C01813=1053.237,59.929,422.366,171.034,32.293,156.055
C01814=1053.230,59.680,422.384,171.032,32.290,156.054
C01815=1053.224,59.431,422.401,171.030,32.288,156.054
C01816=1053.217,59.181,422.419,171.029,32.286,156.054
C01817=1053.211,58.932,422.435,171.027,32.284,156.053
C01818=1053.205,58.682,422.453,171.025,32.282,156.053
C01819=1053.199,58.433,422.470,171.024,32.280,156.053
C01820=1053.193,58.184,422.488,171.022,32.278,156.052
C01821=1053.187,57.935,422.505,171.020,32.276,156.052
C01822=1053.180,57.685,422.522,171.019,32.273,156.052
C01823=1053.174,57.436,422.539,171.017,32.271,156.051
C01824=1053.168,57.186,422.556,171.015,32.269,156.051
C01825=1053.162,56.937,422.574,171.014,32.267,156.051
C01826=1053.155,56.688,422.591,171.012,32.264,156.050
C01827=1053.149,56.439,422.608,171.010,32.262,156.050
C01828=1053.143,56.189,422.625,171.010,32.260,156.050
C01829=1053.137,55.940,422.642,171.008,32.258,156.049
C01830=1053.131,55.690,422.660,171.006,32.256,156.049
C01831=1053.125,55.442,422.677,171.005,32.254,156.049
C01832=1053.118,55.191,422.694,171.003,32.252,156.048
C01833=1053.113,54.942,422.711,171.001,32.250,156.048
C01834=1053.106,54.694,422.728,171.000,32.247,156.048
C01835=1053.099,54.444,422.746,170.998,32.245,156.047
C01836=1053.094,54.195,422.762,170.996,32.243,156.047
C01837=1053.087,53.945,422.780,170.995,32.241,156.047
C01838=1053.082,53.696,422.797,170.993,32.238,156.046
C01839=1053.075,53.446,422.814,170.991,32.236,156.046
C01840=1053.069,53.197,422.831,170.990,32.234,156.046
C01841=1053.063,52.948,422.849,170.988,32.232,156.045
C01842=1053.057,52.699,422.866,170.987,32.230,156.045
C01843=1053.051,52.450,422.882,170.986,32.228,156.045
C01844=1053.045,52.200,422.900,170.984,32.226,156.044
C01845=1053.039,51.950,422.916,170.983,32.223,156.044
C01846=1053.032,51.701,422.934,170.981,32.221,156.044
C01847=1053.026,51.452,422.951,170.979,32.219,156.043
C01848=1053.020,51.203,422.967,170.978,32.216,156.043
C01849=1053.013,50.953,422.985,170.976,32.214,156.043
C01850=1053.008,50.704,423.002,170.974,32.212,156.042
C01851=1053.002,50.455,423.019,170.973,32.210,156.042
C01852=1052.995,50.205,423.036,170.971,32.208,156.041
C01853=1052.990,49.956,423.053,170.969,32.206,156.041
C01854=1052.983,49.706,423.070,170.968,32.204,156.041
C01855=1052.977,49.457,423.086,170.966,32.201,156.040
C01856=1052.972,49.208,423.104,170.964,32.199,156.040
C01857=1052.965,48.958,423.121,170.964,32.197,156.040
C01858=1052.959,48.709,423.138,170.962,32.195,156.040
C01859=1052.953,48.460,423.155,170.960,32.192,156.039
C01860=1052.947,48.210,423.172,170.959,32.190,156.039
C01861=1052.940,47.961,423.189,170.957,32.188,156.039
C01862=1052.935,47.712,423.206,170.955,32.186,156.038
C01863=1052.928,47.462,423.223,170.954,32.184,156.038
C01864=1052.922,47.213,423.239,170.952,32.182,156.037
C01865=1052.917,46.964,423.257,170.950,32.179,156.037
C01866=1052.911,46.714,423.273,170.949,32.177,156.037
C01867=1052.904,46.465,423.290,170.947,32.175,156.036
C01868=1052.899,46.215,423.307,170.945,32.173,156.036
C01869=1052.891,45.930,423.327,170.944,32.170,156.036
C01870=1052.885,45.644,423.345,170.942,32.168,156.035
C01871=1052.877,45.358,423.365,170.941,32.165,156.035
C01872=1052.870,45.072,423.385,170.939,32.162,156.034
C01873=1052.864,44.823,423.401,170.937,32.160,156.034
C01874=1052.859,44.573,423.418,170.936,32.158,156.034
C01875=1052.853,44.325,423.435,170.934,32.156,156.033
C01876=1052.846,44.075,423.451,170.932,32.154,156.033
C01877=1052.841,43.826,423.469,170.931,32.152,156.033
C01878=1052.835,43.576,423.485,170.929,32.149,156.032
C01879=1052.828,43.326,423.502,170.927,32.147,156.032
C01880=1052.822,43.077,423.519,170.926,32.145,156.032
C01881=1052.816,42.828,423.535,170.924,32.143,156.032
C01882=1052.810,42.579,423.551,170.922,32.141,156.031
C01883=1052.803,42.329,423.569,170.921,32.138,156.031
C01884=1052.797,42.080,423.585,170.920,32.136,156.030
C01885=1052.791,41.831,423.601,170.918,32.134,156.030
C01886=1052.785,41.581,423.619,170.917,32.132,156.030
C01887=1052.779,41.332,423.635,170.915,32.130,156.030
C01888=1052.773,41.082,423.651,170.913,32.128,156.029
C01889=1052.767,40.833,423.669,170.911,32.125,156.029
C01890=1052.761,40.583,423.685,170.910,32.123,156.029
C01891=1052.755,40.334,423.701,170.908,32.121,156.028
C01892=1052.749,40.085,423.718,170.906,32.119,156.028
C01893=1052.743,39.836,423.735,170.905,32.117,156.028
C01894=1052.736,39.586,423.751,170.903,32.115,156.027
C01895=1052.730,39.337,423.768,170.901,32.113,156.027
C01896=1052.724,39.087,423.784,170.900,32.111,156.027
C01897=1052.718,38.838,423.800,170.899,32.109,156.026
C01898=1052.712,38.589,423.817,170.897,32.106,156.026
C01899=1052.705,38.339,423.834,170.896,32.104,156.026
C01900=1052.699,38.090,423.850,170.894,32.102,156.025
C01901=1052.693,37.840,423.866,170.892,32.100,156.025
C01902=1052.687,37.591,423.882,170.891,32.098,156.025
C01903=1052.681,37.342,423.900,170.889,32.096,156.024
C01904=1052.675,37.092,423.916,170.887,32.093,156.024
C01905=1052.669,36.843,423.932,170.886,32.091,156.024
C01906=1052.662,36.594,423.948,170.884,32.089,156.023
C01907=1052.656,36.345,423.964,170.882,32.087,156.023
C01908=1052.649,36.094,423.981,170.881,32.085,156.023
C01909=1052.644,35.845,423.997,170.879,32.083,156.022
C01910=1052.638,35.596,424.013,170.878,32.081,156.022
C01911=1052.632,35.346,424.030,170.876,32.079,156.022
C01912=1052.624,35.097,424.046,170.875,32.077,156.022
C01913=1052.618,34.848,424.063,170.873,32.075,156.021
C01914=1052.612,34.599,424.079,170.871,32.072,156.021
C01915=1052.606,34.349,424.095,170.870,32.070,156.021
C01916=1052.600,34.100,424.111,170.868,32.068,156.020
C01917=1052.594,33.851,424.127,170.866,32.066,156.020
C01918=1052.587,33.601,424.144,170.865,32.064,156.020
C01919=1052.581,33.351,424.160,170.863,32.062,156.019
C01920=1052.575,33.102,424.176,170.861,32.060,156.019
C01921=1052.569,32.853,424.192,170.860,32.058,156.019
C01922=1052.563,32.603,424.209,170.858,32.056,156.018
C01923=1052.556,32.354,424.224,170.857,32.053,156.018
C01924=1052.550,32.104,424.241,170.855,32.051,156.018
C01925=1052.544,31.855,424.257,170.854,32.049,156.017
C01926=1052.538,31.606,424.273,170.852,32.047,156.017
C01927=1052.532,31.356,424.290,170.850,32.045,156.017
C01928=1052.525,31.107,424.305,170.849,32.043,156.017
C01929=1052.519,30.858,424.322,170.847,32.041,156.016
C01930=1052.513,30.609,424.338,170.845,32.039,156.016
C01931=1052.508,30.359,424.354,170.844,32.037,156.015
C01932=1052.501,30.109,424.371,170.842,32.035,156.015
C01933=1052.494,29.824,424.389,170.840,32.032,156.015
C01934=1052.487,29.538,424.407,170.838,32.030,156.014
C01935=1052.480,29.252,424.426,170.837,32.028,156.014
C01936=1052.474,28.966,424.444,170.835,32.025,156.014
C01937=1052.467,28.717,424.459,170.833,32.023,156.014
C01938=1052.461,28.467,424.475,170.832,32.021,156.013
C01939=1052.454,28.217,424.492,170.830,32.019,156.013
C01940=1052.448,27.968,424.508,170.828,32.017,156.013
C01941=1052.442,27.719,424.524,170.827,32.015,156.012
C01942=1052.436,27.470,424.540,170.825,32.013,156.012
C01943=1052.429,27.220,424.555,170.823,32.011,156.012
C01944=1052.423,26.971,424.571,170.821,32.009,156.011
C01945=1052.417,26.721,424.588,170.820,32.006,156.011
C01946=1052.411,26.472,424.603,170.818,32.004,156.011
C01947=1052.405,26.223,424.620,170.817,32.002,156.010
C01948=1052.398,25.973,424.635,170.816,32.000,156.010
C01949=1052.392,25.723,424.651,170.814,31.998,156.010
C01950=1052.385,25.474,424.667,170.812,31.996,156.009
C01951=1052.379,25.225,424.683,170.810,31.994,156.009
C01952=1052.374,24.975,424.699,170.809,31.992,156.009
C01953=1052.367,24.726,424.714,170.807,31.990,156.009
C01954=1052.361,24.476,424.731,170.805,31.988,156.008
C01955=1052.354,24.227,424.746,170.804,31.986,156.008
C01956=1052.349,23.977,424.762,170.802,31.984,156.008
C01957=1052.342,23.728,424.777,170.800,31.982,156.007
C01958=1052.336,23.479,424.794,170.798,31.979,156.007
C01959=1052.330,23.229,424.809,170.798,31.978,156.007
C01960=1052.324,22.980,424.825,170.796,31.975,156.006
C01961=1052.318,22.731,424.841,170.794,31.973,156.006
C01962=1052.311,22.481,424.856,170.793,31.971,156.006
C01963=1052.305,22.232,424.872,170.791,31.969,156.006
C01964=1052.299,21.983,424.888,170.789,31.967,156.005
C01965=1052.293,21.733,424.904,170.787,31.965,156.005
C01966=1052.286,21.484,424.919,170.786,31.963,156.005
C01967=1052.280,21.234,424.936,170.784,31.961,156.004
C01968=1052.275,20.984,424.951,170.782,31.959,156.004
C01969=1052.268,20.735,424.967,170.781,31.957,156.004
C01970=1052.262,20.485,424.982,170.779,31.955,156.003
C01971=1052.256,20.236,424.998,170.778,31.953,156.003
C01972=1052.250,19.987,425.014,170.776,31.951,156.003
C01973=1052.243,19.737,425.029,170.775,31.949,156.003
C01974=1052.237,19.488,425.045,170.773,31.947,156.002
C01975=1052.231,19.238,425.060,170.771,31.945,156.002
C01976=1052.224,18.989,425.076,170.769,31.943,156.002
C01977=1052.219,18.739,425.092,170.768,31.941,156.001
C01978=1052.212,18.490,425.107,170.766,31.939,156.001
C01979=1052.206,18.240,425.123,170.764,31.937,156.001
C01980=1052.200,17.991,425.138,170.762,31.934,156.001
C01981=1052.193,17.741,425.153,170.761,31.933,156.000
C01982=1052.187,17.492,425.170,170.760,31.930,156.000
C01983=1052.181,17.242,425.185,170.758,31.928,156.000
C01984=1052.175,16.993,425.201,170.757,31.926,155.999
C01985=1052.169,16.743,425.216,170.755,31.924,155.999
C01986=1052.162,16.494,425.231,170.753,31.922,155.999
C01987=1052.156,16.244,425.247,170.751,31.920,155.998
C01988=1052.150,15.996,425.262,170.750,31.918,155.998
C01989=1052.144,15.746,425.277,170.748,31.916,155.998
C01990=1052.138,15.497,425.293,170.746,31.914,155.998
C01991=1052.131,15.247,425.308,170.744,31.913,155.997
C01992=1052.126,14.998,425.325,170.743,31.911,155.997
C01993=1052.119,14.748,425.340,170.741,31.909,155.997
C01994=1052.113,14.499,425.355,170.740,31.906,155.996
C01995=1052.107,14.249,425.371,170.738,31.904,155.996
C01996=1052.100,14.000,425.386,170.737,31.902,155.996
C01997=1052.094,13.715,425.403,170.735,31.900,155.996
C01998=1052.087,13.431,425.420,170.733,31.898,155.995
C01999=1052.079,13.146,425.439,170.731,31.896,155.995
C02000=1052.071,12.862,425.455,170.729,31.893,155.995
C02001=1052.065,12.612,425.471,170.727,31.891,155.994
C02002=1052.059,12.362,425.486,170.725,31.889,155.994
C02003=1052.052,12.113,425.502,170.723,31.887,155.994
C02004=1052.046,11.864,425.517,170.722,31.886,155.994
C02005=1052.040,11.615,425.531,170.721,31.884,155.993
C02006=1052.034,11.365,425.546,170.719,31.882,155.993
C02007=1052.027,11.116,425.562,170.717,31.880,155.993
C02008=1052.021,10.866,425.577,170.715,31.877,155.992
C02009=1052.015,10.616,425.592,170.714,31.876,155.992
C02010=1052.009,10.367,425.607,170.712,31.874,155.992
C02011=1052.002,10.118,425.623,170.710,31.872,155.992
C02012=1051.996,9.868,425.638,170.708,31.870,155.991
C02013=1051.989,9.618,425.653,170.707,31.868,155.991
C02014=1051.983,9.369,425.667,170.705,31.866,155.991
C02015=1051.977,9.120,425.684,170.703,31.864,155.990
C02016=1051.971,8.870,425.699,170.702,31.862,155.990
C02017=1051.965,8.621,425.713,170.701,31.860,155.990
C02018=1051.958,8.371,425.728,170.699,31.858,155.990
C02019=1051.952,8.121,425.743,170.697,31.856,155.989
C02020=1051.945,7.872,425.759,170.695,31.854,155.989
C02021=1051.939,7.623,425.774,170.693,31.852,155.989
C02022=1051.933,7.374,425.789,170.692,31.851,155.989
C02023=1051.927,7.124,425.803,170.690,31.848,155.988
C02024=1051.921,6.874,425.819,170.688,31.846,155.988
C02025=1051.915,6.625,425.834,170.686,31.844,155.988
C02026=1051.909,6.376,425.849,170.685,31.842,155.987
C02027=1051.902,6.127,425.864,170.684,31.840,155.987
C02028=1051.896,5.877,425.879,170.682,31.839,155.987
C02029=1051.889,5.627,425.894,170.680,31.837,155.987
C02030=1051.883,5.378,425.909,170.678,31.835,155.986
C02031=1051.877,5.129,425.924,170.677,31.833,155.986
C02032=1051.871,4.879,425.939,170.675,31.831,155.986
C02033=1051.865,4.629,425.954,170.673,31.828,155.985
C02034=1051.859,4.379,425.969,170.671,31.827,155.985
C02035=1051.853,4.130,425.984,170.670,31.825,155.985
C02036=1051.847,3.881,425.999,170.668,31.823,155.985
C02037=1051.840,3.631,426.014,170.666,31.821,155.984
C02038=1051.834,3.381,426.028,170.665,31.819,155.984
C02039=1051.828,3.132,426.043,170.663,31.817,155.984
C02040=1051.821,2.883,426.059,170.662,31.815,155.984
C02041=1051.815,2.634,426.074,170.660,31.813,155.983
C02042=1051.809,2.384,426.089,170.658,31.811,155.983
C02043=1051.803,2.135,426.103,170.656,31.809,155.983
C02044=1051.797,1.885,426.118,170.654,31.807,155.982
C02045=1051.790,1.636,426.133,170.653,31.806,155.982
C02046=1051.784,1.386,426.147,170.651,31.803,155.982
C02047=1051.778,1.137,426.162,170.649,31.801,155.982
C02048=1051.772,0.887,426.177,170.648,31.799,155.981
C02049=1051.766,0.637,426.192,170.647,31.797,155.981
C02050=1051.760,0.388,426.207,170.645,31.795,155.981
C02051=1051.754,0.138,426.222,170.643,31.794,155.981
C02052=1051.748,-0.111,426.237,170.641,31.792,155.980
C02053=1051.742,-0.360,426.251,170.639,31.790,155.980
C02054=1051.736,-0.610,426.266,170.638,31.788,155.980
C02055=1051.729,-0.860,426.281,170.636,31.785,155.979
C02056=1051.723,-1.109,426.296,170.634,31.784,155.979
C02057=1051.717,-1.358,426.311,170.632,31.782,155.979
C02058=1051.711,-1.608,426.326,170.630,31.780,155.979
C02059=1051.705,-1.857,426.340,170.630,31.778,155.978
C02060=1051.699,-2.107,426.355,170.628,31.776,155.978
C02061=1051.692,-2.389,426.371,170.626,31.774,155.978
C02062=1051.685,-2.672,426.388,170.624,31.772,155.977
C02063=1051.678,-2.954,426.405,170.622,31.769,155.977
C02064=1051.671,-3.238,426.421,170.620,31.767,155.977
C02065=1051.665,-3.487,426.436,170.618,31.765,155.977
C02066=1051.659,-3.736,426.451,170.616,31.763,155.976
C02067=1051.652,-3.986,426.466,170.614,31.761,155.976
C02068=1051.646,-4.235,426.479,170.612,31.760,155.976
C02069=1051.640,-4.485,426.494,170.611,31.757,155.976
C02070=1051.633,-4.735,426.509,170.610,31.756,155.975
C02071=1051.627,-4.983,426.524,170.608,31.754,155.975
C02072=1051.621,-5.233,426.537,170.606,31.752,155.975
C02073=1051.614,-5.483,426.552,170.604,31.750,155.975
C02074=1051.608,-5.732,426.567,170.602,31.748,155.974
C02075=1051.602,-5.982,426.580,170.601,31.746,155.974
C02076=1051.595,-6.232,426.595,170.599,31.745,155.974
C02077=1051.589,-6.481,426.610,170.597,31.743,155.974
C02078=1051.583,-6.730,426.625,170.595,31.741,155.973
C02079=1051.577,-6.980,426.638,170.594,31.739,155.973
C02080=1051.570,-7.229,426.653,170.592,31.737,155.973
C02081=1051.564,-7.479,426.668,170.591,31.736,155.973
C02082=1051.559,-7.728,426.682,170.589,31.734,155.972
C02083=1051.552,-7.978,426.696,170.587,31.732,155.972
C02084=1051.545,-8.227,426.711,170.585,31.730,155.972
C02085=1051.540,-8.477,426.725,170.583,31.728,155.972
C02086=1051.533,-8.726,426.739,170.581,31.726,155.971
C02087=1051.527,-8.976,426.753,170.579,31.724,155.971
C02088=1051.521,-9.226,426.768,170.578,31.722,155.971
C02089=1051.515,-9.475,426.783,170.576,31.721,155.971
C02090=1051.508,-9.725,426.796,170.575,31.719,155.970
C02091=1051.502,-9.974,426.811,170.573,31.717,155.970
C02092=1051.496,-10.224,426.825,170.571,31.715,155.970
C02093=1051.489,-10.473,426.840,170.569,31.713,155.970
C02094=1051.483,-10.722,426.854,170.568,31.712,155.969
C02095=1051.477,-10.972,426.868,170.566,31.710,155.969
C02096=1051.471,-11.221,426.882,170.564,31.708,155.969
C02097=1051.465,-11.471,426.897,170.562,31.706,155.969
C02098=1051.459,-11.720,426.911,170.560,31.704,155.968
C02099=1051.452,-11.970,426.925,170.558,31.702,155.968
C02100=1051.446,-12.220,426.940,170.557,31.700,155.968
C02101=1051.440,-12.469,426.954,170.556,31.698,155.968
C02102=1051.433,-12.719,426.968,170.554,31.697,155.967
C02103=1051.428,-12.968,426.982,170.552,31.695,155.967
C02104=1051.421,-13.218,426.997,170.550,31.693,155.967
C02105=1051.415,-13.467,427.010,170.548,31.691,155.967
C02106=1051.409,-13.717,427.025,170.546,31.689,155.966
C02107=1051.403,-13.966,427.039,170.545,31.688,155.966
C02108=1051.396,-14.216,427.053,170.543,31.686,155.966
C02109=1051.391,-14.465,427.067,170.541,31.684,155.966
C02110=1051.384,-14.716,427.081,170.540,31.682,155.965
C02111=1051.378,-14.964,427.095,170.538,31.680,155.965
C02112=1051.372,-15.215,427.110,170.536,31.678,155.965
C02113=1051.365,-15.463,427.124,170.534,31.676,155.965
C02114=1051.359,-15.714,427.138,170.532,31.675,155.965
C02115=1051.353,-15.963,427.151,170.531,31.673,155.964
C02116=1051.347,-16.212,427.166,170.529,31.671,155.964
C02117=1051.340,-16.462,427.179,170.527,31.669,155.964
C02118=1051.334,-16.712,427.194,170.525,31.668,155.964
C02119=1051.328,-16.961,427.208,170.523,31.666,155.963
C02120=1051.322,-17.211,427.222,170.522,31.664,155.963
C02121=1051.316,-17.460,427.235,170.520,31.663,155.963
C02122=1051.308,-17.710,427.249,170.518,31.661,155.963
C02123=1051.303,-17.959,427.263,170.517,31.659,155.962
C02124=1051.297,-18.208,427.277,170.515,31.657,155.962
C02125=1051.290,-18.489,427.292,170.513,31.656,155.962
C02126=1051.283,-18.771,427.308,170.510,31.653,155.962
C02127=1051.276,-19.052,427.324,170.508,31.651,155.961
C02128=1051.269,-19.333,427.339,170.506,31.649,155.961
C02129=1051.262,-19.582,427.354,170.504,31.648,155.961
C02130=1051.256,-19.831,427.367,170.503,31.646,155.961
C02131=1051.250,-20.082,427.381,170.501,31.644,155.961
C02132=1051.243,-20.331,427.395,170.500,31.643,155.960
C02133=1051.237,-20.581,427.410,170.498,31.641,155.960
C02134=1051.231,-20.830,427.423,170.496,31.639,155.960
C02135=1051.225,-21.079,427.436,170.494,31.637,155.960
C02136=1051.219,-21.329,427.450,170.492,31.635,155.959
C02137=1051.212,-21.578,427.464,170.490,31.633,155.959
C02138=1051.206,-21.828,427.479,170.488,31.632,155.959
C02139=1051.200,-22.078,427.492,170.486,31.630,155.959
C02140=1051.193,-22.327,427.505,170.485,31.628,155.959
C02141=1051.187,-22.577,427.519,170.484,31.627,155.958
C02142=1051.181,-22.826,427.533,170.482,31.625,155.958
C02143=1051.175,-23.075,427.547,170.480,31.623,155.958
C02144=1051.169,-23.325,427.561,170.478,31.621,155.958
C02145=1051.162,-23.575,427.574,170.476,31.620,155.957
C02146=1051.156,-23.825,427.588,170.474,31.618,155.957
C02147=1051.150,-24.074,427.602,170.472,31.616,155.957
C02148=1051.144,-24.323,427.615,170.470,31.615,155.957
C02149=1051.138,-24.574,427.629,170.468,31.612,155.957
C02150=1051.132,-24.823,427.642,170.467,31.611,155.956
C02151=1051.125,-25.072,427.656,170.465,31.609,155.956
C02152=1051.119,-25.322,427.671,170.464,31.607,155.956
C02153=1051.113,-25.571,427.684,170.462,31.606,155.956
C02154=1051.107,-25.821,427.698,170.460,31.604,155.955
C02155=1051.101,-26.070,427.711,170.458,31.602,155.955
C02156=1051.094,-26.320,427.725,170.456,31.601,155.955
C02157=1051.089,-26.569,427.738,170.454,31.599,155.955
C02158=1051.083,-26.819,427.752,170.452,31.597,155.955
C02159=1051.076,-27.069,427.765,170.450,31.596,155.954
C02160=1051.070,-27.318,427.779,170.449,31.594,155.954
C02161=1051.063,-27.567,427.792,170.447,31.592,155.954
C02162=1051.057,-27.818,427.806,170.445,31.591,155.954
C02163=1051.051,-28.067,427.819,170.443,31.589,155.954
C02164=1051.045,-28.316,427.833,170.442,31.587,155.953
C02165=1051.038,-28.566,427.846,170.440,31.586,155.953
C02166=1051.032,-28.815,427.860,170.438,31.584,155.953
C02167=1051.026,-29.065,427.873,170.436,31.583,155.953
C02168=1051.019,-29.315,427.886,170.434,31.581,155.953
C02169=1051.014,-29.565,427.900,170.432,31.579,155.952
C02170=1051.007,-29.814,427.913,170.431,31.578,155.952
C02171=1051.001,-30.064,427.927,170.429,31.576,155.952
C02172=1050.994,-30.313,427.940,170.427,31.574,155.952
C02173=1050.988,-30.562,427.953,170.425,31.572,155.952
C02174=1050.982,-30.812,427.966,170.423,31.571,155.951
C02175=1050.975,-31.062,427.980,170.421,31.569,155.951
C02176=1050.969,-31.311,427.993,170.419,31.568,155.951
C02177=1050.963,-31.561,428.006,170.417,31.566,155.951
C02178=1050.958,-31.810,428.020,170.415,31.564,155.951
C02179=1050.951,-32.060,428.033,170.413,31.563,155.950
C02180=1050.944,-32.310,428.047,170.412,31.561,155.950
C02181=1050.938,-32.559,428.060,170.410,31.560,155.950
C02182=1050.932,-32.808,428.073,170.409,31.558,155.950
C02183=1050.926,-33.059,428.086,170.407,31.556,155.950
C02184=1050.919,-33.308,428.099,170.405,31.555,155.949
C02185=1050.913,-33.557,428.113,170.403,31.553,155.949
C02186=1050.907,-33.807,428.126,170.401,31.551,155.949
C02187=1050.901,-34.056,428.139,170.399,31.550,155.949
C02188=1050.894,-34.306,428.152,170.397,31.548,155.949
C02189=1050.888,-34.587,428.167,170.395,31.547,155.948
C02190=1050.881,-34.867,428.182,170.393,31.544,155.948
C02191=1050.874,-35.147,428.197,170.391,31.543,155.948
C02192=1050.867,-35.427,428.212,170.389,31.541,155.948
C02193=1050.860,-35.676,428.225,170.387,31.539,155.948
C02194=1050.855,-35.926,428.238,170.385,31.538,155.947
C02195=1050.848,-36.175,428.251,170.383,31.536,155.947
C02196=1050.842,-36.425,428.264,170.381,31.535,155.947
C02197=1050.835,-36.675,428.278,170.379,31.533,155.947
C02198=1050.829,-36.925,428.290,170.377,31.531,155.947
C02199=1050.823,-37.174,428.304,170.376,31.530,155.946
C02200=1050.818,-37.423,428.317,170.374,31.528,155.946
C02201=1050.812,-37.673,428.330,170.372,31.527,155.946
C02202=1050.806,-37.923,428.343,170.370,31.525,155.946
C02203=1050.799,-38.172,428.357,170.368,31.523,155.946
C02204=1050.793,-38.422,428.369,170.366,31.521,155.946
C02205=1050.787,-38.672,428.383,170.364,31.520,155.945
C02206=1050.781,-38.922,428.395,170.362,31.518,155.945
C02207=1050.774,-39.170,428.408,170.361,31.517,155.945
C02208=1050.768,-39.420,428.421,170.359,31.516,155.945
C02209=1050.762,-39.670,428.434,170.358,31.514,155.945
C02210=1050.755,-39.920,428.447,170.356,31.513,155.944
C02211=1050.749,-40.169,428.460,170.354,31.511,155.944
C02212=1050.743,-40.419,428.473,170.352,31.510,155.944
C02213=1050.736,-40.668,428.485,170.350,31.508,155.944
C02214=1050.730,-40.918,428.498,170.348,31.507,155.944
C02215=1050.724,-41.167,428.511,170.346,31.505,155.944
C02216=1050.718,-41.417,428.524,170.344,31.504,155.943
C02217=1050.711,-41.667,428.537,170.342,31.502,155.943
C02218=1050.704,-41.916,428.550,170.340,31.501,155.943
C02219=1050.698,-42.166,428.562,170.339,31.499,155.943
C02220=1050.692,-42.415,428.576,170.337,31.498,155.943
C02221=1050.686,-42.665,428.588,170.335,31.496,155.943
C02222=1050.680,-42.915,428.601,170.333,31.495,155.942
C02223=1050.674,-43.164,428.614,170.331,31.493,155.942
C02224=1050.667,-43.413,428.627,170.329,31.491,155.942
C02225=1050.661,-43.663,428.639,170.327,31.490,155.942
C02226=1050.655,-43.913,428.653,170.325,31.488,155.942
C02227=1050.649,-44.162,428.665,170.323,31.487,155.942
C02228=1050.643,-44.412,428.678,170.321,31.485,155.941
C02229=1050.636,-44.661,428.690,170.320,31.484,155.941
C02230=1050.630,-44.912,428.703,170.318,31.482,155.941
C02231=1050.624,-45.161,428.717,170.316,31.481,155.941
C02232=1050.618,-45.411,428.729,170.314,31.479,155.941
C02233=1050.611,-45.660,428.742,170.312,31.479,155.941
C02234=1050.605,-45.910,428.754,170.310,31.477,155.941
C02235=1050.599,-46.160,428.767,170.308,31.476,155.940
C02236=1050.593,-46.409,428.780,170.306,31.474,155.940
C02237=1050.587,-46.659,428.793,170.303,31.472,155.940
C02238=1050.580,-46.908,428.805,170.301,31.471,155.940
C02239=1050.574,-47.158,428.818,170.300,31.469,155.940
C02240=1050.568,-47.408,428.830,170.298,31.468,155.940
C02241=1050.562,-47.657,428.843,170.296,31.466,155.939
C02242=1050.555,-47.906,428.856,170.294,31.465,155.939
C02243=1050.549,-48.156,428.868,170.292,31.463,155.939
C02244=1050.543,-48.406,428.881,170.290,31.462,155.939
C02245=1050.537,-48.656,428.893,170.288,31.460,155.939
C02246=1050.530,-48.905,428.906,170.286,31.459,155.939
C02247=1050.525,-49.155,428.919,170.284,31.457,155.938
C02248=1050.519,-49.404,428.931,170.282,31.456,155.938
C02249=1050.513,-49.653,428.944,170.280,31.455,155.938
C02250=1050.506,-49.903,428.956,170.279,31.453,155.938
C02251=1050.500,-50.153,428.969,170.277,31.452,155.938
C02252=1050.495,-50.403,428.981,170.275,31.450,155.938
C02253=1050.486,-50.684,428.995,170.273,31.449,155.938
C02254=1050.480,-50.964,429.009,170.271,31.447,155.937
C02255=1050.473,-51.245,429.023,170.268,31.446,155.937
C02256=1050.465,-51.526,429.037,170.266,31.444,155.937
C02257=1050.460,-51.775,429.049,170.264,31.443,155.937
C02258=1050.453,-52.025,429.061,170.262,31.442,155.937
C02259=1050.446,-52.274,429.074,170.261,31.440,155.937
C02260=1050.440,-52.524,429.086,170.259,31.439,155.937
C02261=1050.433,-52.773,429.098,170.257,31.438,155.936
C02262=1050.427,-53.023,429.111,170.255,31.436,155.936
C02263=1050.421,-53.273,429.123,170.253,31.435,155.936
C02264=1050.415,-53.523,429.135,170.251,31.434,155.936
C02265=1050.408,-53.772,429.147,170.248,31.432,155.936
C02266=1050.402,-54.022,429.159,170.246,31.431,155.936
C02267=1050.396,-54.272,429.172,170.244,31.430,155.936
C02268=1050.389,-54.521,429.184,170.242,31.428,155.935
C02269=1050.383,-54.771,429.196,170.240,31.427,155.935
C02270=1050.376,-55.020,429.209,170.239,31.426,155.935
C02271=1050.370,-55.269,429.221,170.237,31.424,155.935
C02272=1050.364,-55.519,429.233,170.235,31.423,155.935
C02273=1050.358,-55.769,429.245,170.233,31.422,155.935
C02274=1050.352,-56.018,429.258,170.231,31.421,155.935
C02275=1050.345,-56.268,429.270,170.229,31.420,155.935
C02276=1050.338,-56.518,429.282,170.227,31.418,155.934
C02277=1050.332,-56.767,429.294,170.225,31.417,155.934
C02278=1050.326,-57.017,429.306,170.223,31.416,155.934
C02279=1050.319,-57.267,429.318,170.221,31.414,155.934
C02280=1050.314,-57.517,429.330,170.219,31.413,155.934
C02281=1050.308,-57.766,429.341,170.217,31.412,155.934
C02282=1050.302,-58.016,429.354,170.215,31.411,155.934
C02283=1050.295,-58.265,429.366,170.213,31.409,155.934
C02284=1050.288,-58.515,429.378,170.211,31.408,155.934
C02285=1050.282,-58.765,429.390,170.209,31.407,155.933
C02286=1050.276,-59.014,429.402,170.207,31.405,155.933
C02287=1050.269,-59.264,429.414,170.205,31.404,155.933
C02288=1050.264,-59.513,429.427,170.203,31.403,155.933
C02289=1050.257,-59.763,429.439,170.201,31.402,155.933
C02290=1050.251,-60.012,429.450,170.199,31.400,155.933
C02291=1050.245,-60.262,429.463,170.198,31.399,155.933
C02292=1050.238,-60.512,429.474,170.196,31.398,155.933
C02293=1050.232,-60.761,429.486,170.194,31.396,155.932
C02294=1050.226,-61.011,429.498,170.191,31.395,155.932
C02295=1050.220,-61.261,429.510,170.189,31.394,155.932
C02296=1050.214,-61.511,429.523,170.187,31.393,155.932
C02297=1050.207,-61.760,429.535,170.185,31.391,155.932
C02298=1050.201,-62.010,429.546,170.183,31.390,155.932
C02299=1050.196,-62.260,429.558,170.181,31.389,155.932
C02300=1050.189,-62.509,429.570,170.179,31.387,155.932
C02301=1050.182,-62.759,429.582,170.178,31.387,155.932
C02302=1050.176,-63.008,429.594,170.176,31.385,155.931
C02303=1050.171,-63.258,429.606,170.174,31.384,155.931
C02304=1050.164,-63.508,429.618,170.172,31.383,155.931
C02305=1050.157,-63.757,429.630,170.169,31.382,155.931
C02306=1050.151,-64.007,429.642,170.167,31.380,155.931
C02307=1050.146,-64.257,429.653,170.165,31.379,155.931
C02308=1050.139,-64.506,429.665,170.163,31.378,155.931
C02309=1050.133,-64.756,429.678,170.161,31.377,155.931
C02310=1050.127,-65.005,429.689,170.159,31.375,155.931
C02311=1050.121,-65.255,429.700,170.157,31.374,155.931
C02312=1050.115,-65.505,429.713,170.156,31.373,155.930
C02313=1050.108,-65.755,429.725,170.154,31.372,155.930
C02314=1050.102,-66.003,429.736,170.152,31.370,155.930
C02315=1050.096,-66.254,429.748,170.150,31.370,155.930
C02316=1050.090,-66.504,429.760,170.147,31.368,155.930
C02317=1050.083,-66.785,429.774,170.145,31.367,155.930
C02318=1050.076,-67.067,429.786,170.143,31.365,155.930
C02319=1050.069,-67.349,429.800,170.140,31.364,155.930
C02320=1050.062,-67.631,429.813,170.138,31.363,155.930
C02321=1050.056,-67.881,429.824,170.136,31.361,155.929
C02322=1050.050,-68.131,429.837,170.135,31.360,155.929
C02323=1050.044,-68.381,429.848,170.133,31.359,155.929
C02324=1050.038,-68.630,429.860,170.131,31.358,155.929
C02325=1050.031,-68.879,429.872,170.128,31.356,155.929
C02326=1050.026,-69.129,429.883,170.126,31.355,155.929
C02327=1050.019,-69.379,429.895,170.124,31.354,155.929
C02328=1050.013,-69.629,429.906,170.122,31.353,155.929
C02329=1050.007,-69.878,429.918,170.120,31.352,155.929
C02330=1050.001,-70.128,429.931,170.118,31.351,155.929
C02331=1049.995,-70.378,429.942,170.116,31.350,155.928
C02332=1049.989,-70.627,429.953,170.115,31.348,155.928
C02333=1049.982,-70.877,429.965,170.113,31.347,155.928
C02334=1049.977,-71.126,429.977,170.110,31.346,155.928
C02335=1049.971,-71.376,429.988,170.108,31.345,155.928
C02336=1049.965,-71.625,430.000,170.106,31.344,155.928
C02337=1049.958,-71.875,430.011,170.104,31.342,155.928
C02338=1049.953,-72.125,430.023,170.102,31.341,155.928
C02339=1049.947,-72.375,430.034,170.100,31.340,155.928
C02340=1049.940,-72.624,430.046,170.098,31.339,155.928
C02341=1049.934,-72.874,430.057,170.096,31.338,155.928
C02342=1049.928,-73.124,430.070,170.094,31.337,155.927
C02343=1049.923,-73.373,430.081,170.092,31.335,155.927
C02344=1049.916,-73.623,430.092,170.090,31.334,155.927
C02345=1049.910,-73.872,430.103,170.088,31.333,155.927
C02346=1049.904,-74.122,430.115,170.086,31.332,155.927
C02347=1049.897,-74.372,430.127,170.084,31.331,155.927
C02348=1049.892,-74.621,430.137,170.082,31.330,155.927
C02349=1049.885,-74.872,430.149,170.080,31.329,155.927
C02350=1049.879,-75.121,430.160,170.078,31.328,155.927
C02351=1049.873,-75.371,430.172,170.075,31.327,155.927
C02352=1049.866,-75.620,430.184,170.073,31.326,155.927
C02353=1049.861,-75.870,430.194,170.071,31.324,155.926
C02354=1049.854,-76.120,430.206,170.070,31.324,155.926
C02355=1049.848,-76.369,430.217,170.068,31.323,155.926
C02356=1049.842,-76.619,430.228,170.066,31.322,155.926
C02357=1049.836,-76.869,430.239,170.064,31.321,155.926
C02358=1049.829,-77.118,430.251,170.061,31.320,155.926
C02359=1049.824,-77.368,430.262,170.059,31.318,155.926
C02360=1049.817,-77.618,430.273,170.057,31.317,155.926
C02361=1049.812,-77.867,430.284,170.055,31.316,155.926
C02362=1049.805,-78.117,430.296,170.053,31.316,155.926
C02363=1049.799,-78.366,430.307,170.051,31.315,155.926
C02364=1049.793,-78.617,430.318,170.049,31.314,155.926
C02365=1049.787,-78.866,430.329,170.047,31.312,155.926
C02366=1049.780,-79.116,430.341,170.045,31.311,155.926
C02367=1049.775,-79.365,430.352,170.043,31.310,155.926
C02368=1049.768,-79.615,430.363,170.041,31.309,155.926
C02369=1049.762,-79.864,430.374,170.039,31.308,155.925
C02370=1049.756,-80.115,430.385,170.037,31.308,155.925
C02371=1049.750,-80.363,430.396,170.034,31.306,155.925
C02372=1049.743,-80.614,430.408,170.032,31.306,155.925
C02373=1049.737,-80.863,430.418,170.030,31.305,155.925
C02374=1049.730,-81.113,430.429,170.028,31.304,155.925
C02375=1049.725,-81.363,430.440,170.026,31.303,155.925
C02376=1049.718,-81.613,430.451,170.024,31.302,155.925
C02377=1049.712,-81.861,430.462,170.022,31.301,155.925
C02378=1049.705,-82.111,430.474,170.020,31.300,155.925
C02379=1049.699,-82.361,430.484,170.018,31.299,155.925
C02380=1049.692,-82.611,430.495,170.016,31.298,155.925
C02381=1049.685,-82.895,430.508,170.013,31.297,155.925
C02382=1049.679,-83.180,430.520,170.011,31.296,155.925
C02383=1049.672,-83.464,430.532,170.008,31.295,155.925
C02384=1049.665,-83.748,430.545,170.006,31.294,155.925
C02385=1049.658,-83.998,430.556,170.004,31.293,155.925
C02386=1049.652,-84.247,430.567,170.002,31.292,155.925
C02387=1049.645,-84.497,430.578,169.999,31.291,155.925
C02388=1049.640,-84.747,430.589,169.998,31.291,155.925
C02389=1049.633,-84.996,430.599,169.996,31.290,155.925
C02390=1049.627,-85.246,430.610,169.994,31.289,155.925
C02391=1049.621,-85.495,430.621,169.992,31.288,155.925
C02392=1049.615,-85.746,430.632,169.990,31.288,155.925
C02393=1049.608,-85.995,430.643,169.987,31.286,155.925
C02394=1049.602,-86.245,430.654,169.985,31.286,155.924
C02395=1049.596,-86.495,430.665,169.983,31.285,155.924
C02396=1049.590,-86.744,430.675,169.981,31.284,155.924
C02397=1049.583,-86.994,430.686,169.979,31.283,155.924
C02398=1049.578,-87.243,430.697,169.976,31.282,155.924
C02399=1049.571,-87.493,430.707,169.974,31.281,155.924
C02400=1049.565,-87.743,430.719,169.972,31.281,155.924
C02401=1049.559,-87.992,430.729,169.971,31.280,155.924
C02402=1049.552,-88.242,430.740,169.969,31.279,155.924
C02403=1049.546,-88.492,430.751,169.967,31.278,155.924
C02404=1049.540,-88.741,430.762,169.964,31.277,155.924
C02405=1049.534,-88.992,430.772,169.962,31.277,155.924
C02406=1049.528,-89.241,430.783,169.960,31.276,155.924
C02407=1049.522,-89.491,430.794,169.958,31.275,155.924
C02408=1049.515,-89.740,430.804,169.956,31.274,155.924
C02409=1049.509,-89.990,430.815,169.953,31.273,155.924
C02410=1049.503,-90.239,430.825,169.951,31.272,155.924
C02411=1049.497,-90.489,430.837,169.949,31.272,155.924
C02412=1049.491,-90.739,430.847,169.947,31.271,155.924
C02413=1049.485,-90.989,430.857,169.946,31.270,155.924
C02414=1049.479,-91.238,430.868,169.943,31.269,155.924
C02415=1049.473,-91.488,430.879,169.941,31.268,155.924
C02416=1049.466,-91.737,430.889,169.939,31.267,155.924
C02417=1049.460,-91.987,430.900,169.937,31.267,155.924
C02418=1049.454,-92.238,430.911,169.935,31.266,155.924
C02419=1049.448,-92.487,430.921,169.932,31.265,155.924
C02420=1049.442,-92.736,430.932,169.930,31.264,155.924
C02421=1049.436,-92.986,430.942,169.928,31.263,155.924
C02422=1049.430,-93.236,430.953,169.926,31.263,155.924
C02423=1049.424,-93.486,430.964,169.924,31.262,155.924
C02424=1049.417,-93.735,430.974,169.922,31.261,155.924
C02425=1049.412,-93.985,430.985,169.920,31.260,155.924
C02426=1049.405,-94.235,430.995,169.918,31.259,155.924
C02427=1049.399,-94.485,431.006,169.916,31.259,155.924
C02428=1049.393,-94.734,431.017,169.914,31.258,155.924
C02429=1049.387,-94.983,431.027,169.912,31.257,155.924
C02430=1049.382,-95.233,431.037,169.909,31.256,155.924
C02431=1049.374,-95.483,431.048,169.907,31.256,155.924
C02432=1049.369,-95.733,431.059,169.905,31.255,155.924
C02433=1049.363,-95.983,431.069,169.903,31.254,155.924
C02434=1049.357,-96.232,431.079,169.901,31.254,155.924
C02435=1049.351,-96.481,431.090,169.898,31.253,155.924
C02436=1049.344,-96.732,431.100,169.896,31.252,155.924
C02437=1049.339,-96.981,431.111,169.894,31.252,155.924
C02438=1049.332,-97.231,431.120,169.893,31.251,155.924
C02439=1049.327,-97.481,431.131,169.890,31.250,155.924
C02440=1049.320,-97.730,431.141,169.888,31.249,155.924
C02441=1049.314,-97.981,431.152,169.886,31.248,155.924
C02442=1049.308,-98.230,431.162,169.884,31.248,155.924
C02443=1049.302,-98.480,431.172,169.882,31.247,155.924
C02444=1049.296,-98.729,431.183,169.879,31.247,155.924
C02445=1049.288,-99.016,431.195,169.877,31.246,155.924
C02446=1049.281,-99.302,431.206,169.874,31.245,155.924
C02447=1049.274,-99.589,431.217,169.872,31.245,155.924
C02448=1049.268,-99.876,431.230,169.869,31.243,155.924
C02449=1049.261,-100.125,431.240,169.867,31.243,155.924
C02450=1049.255,-100.374,431.249,169.865,31.242,155.924
C02451=1049.249,-100.625,431.261,169.863,31.242,155.924
C02452=1049.242,-100.874,431.270,169.861,31.242,155.924
C02453=1049.236,-101.124,431.281,169.859,31.241,155.924
C02454=1049.230,-101.374,431.291,169.857,31.240,155.924
C02455=1049.224,-101.623,431.301,169.855,31.239,155.924
C02456=1049.218,-101.873,431.311,169.852,31.239,155.924
C02457=1049.212,-102.122,431.321,169.850,31.238,155.924
C02458=1049.205,-102.373,431.331,169.848,31.238,155.924
C02459=1049.199,-102.623,431.341,169.846,31.237,155.924
C02460=1049.193,-102.872,431.352,169.843,31.236,155.924
C02461=1049.187,-103.122,431.361,169.841,31.236,155.924
C02462=1049.181,-103.371,431.372,169.839,31.235,155.924
C02463=1049.175,-103.621,431.381,169.837,31.235,155.924
C02464=1049.169,-103.871,431.391,169.835,31.234,155.924
C02465=1049.163,-104.120,431.402,169.833,31.234,155.924
C02466=1049.156,-104.370,431.411,169.831,31.233,155.924
C02467=1049.151,-104.619,431.422,169.829,31.232,155.924
C02468=1049.144,-104.870,431.432,169.827,31.232,155.924
C02469=1049.138,-105.120,431.442,169.824,31.231,155.924
C02470=1049.131,-105.369,431.452,169.822,31.231,155.924
C02471=1049.126,-105.619,431.462,169.820,31.231,155.924
C02472=1049.120,-105.869,431.472,169.818,31.230,155.924
C02473=1049.113,-106.118,431.482,169.815,31.229,155.924
C02474=1049.107,-106.368,431.492,169.813,31.229,155.924
C02475=1049.102,-106.618,431.502,169.811,31.228,155.924
C02476=1049.095,-106.868,431.511,169.809,31.228,155.924
C02477=1049.089,-107.117,431.522,169.806,31.227,155.924
C02478=1049.083,-107.367,431.531,169.804,31.226,155.924
C02479=1049.077,-107.617,431.541,169.803,31.226,155.924
C02480=1049.071,-107.866,431.552,169.801,31.226,155.924
C02481=1049.065,-108.116,431.561,169.798,31.225,155.925
C02482=1049.059,-108.365,431.571,169.796,31.225,155.925
C02483=1049.052,-108.615,431.580,169.794,31.224,155.925
C02484=1049.046,-108.865,431.590,169.792,31.224,155.925
C02485=1049.040,-109.114,431.600,169.789,31.223,155.925
C02486=1049.034,-109.364,431.610,169.787,31.223,155.925
C02487=1049.027,-109.614,431.619,169.785,31.222,155.925
C02488=1049.022,-109.864,431.629,169.783,31.222,155.925
C02489=1049.016,-110.114,431.639,169.780,31.222,155.925
C02490=1049.009,-110.363,431.649,169.778,31.221,155.925
C02491=1049.003,-110.613,431.659,169.776,31.221,155.925
C02492=1048.997,-110.863,431.668,169.774,31.221,155.925
C02493=1048.991,-111.112,431.678,169.771,31.220,155.925
C02494=1048.985,-111.362,431.687,169.770,31.219,155.925
C02495=1048.978,-111.612,431.697,169.768,31.219,155.925
C02496=1048.972,-111.862,431.707,169.766,31.219,155.925
C02497=1048.966,-112.112,431.716,169.763,31.218,155.925
C02498=1048.960,-112.361,431.727,169.761,31.218,155.925
C02499=1048.954,-112.611,431.737,169.759,31.218,155.925
C02500=1048.948,-112.861,431.746,169.757,31.217,155.925
C02501=1048.942,-113.110,431.756,169.754,31.216,155.925
C02502=1048.936,-113.360,431.765,169.752,31.216,155.926
C02503=1048.929,-113.610,431.775,169.750,31.216,155.926
C02504=1048.923,-113.860,431.784,169.748,31.216,155.926
C02505=1048.917,-114.110,431.794,169.745,31.215,155.926
C02506=1048.911,-114.359,431.804,169.743,31.215,155.926
C02507=1048.905,-114.609,431.813,169.741,31.215,155.926
C02508=1048.899,-114.859,431.823,169.739,31.214,155.926
C02509=1048.891,-115.144,431.833,169.736,31.214,155.926
C02510=1048.885,-115.429,431.845,169.734,31.213,155.926
C02511=1048.877,-115.715,431.856,169.732,31.213,155.926
C02512=1048.870,-116.000,431.866,169.729,31.213,155.926
C02513=1048.864,-116.250,431.876,169.727,31.212,155.926
C02514=1048.858,-116.499,431.885,169.725,31.212,155.926
C02515=1048.852,-116.749,431.895,169.722,31.212,155.926
C02516=1048.846,-116.998,431.904,169.720,31.211,155.927
C02517=1048.840,-117.249,431.913,169.718,31.211,155.927
C02518=1048.834,-117.499,431.923,169.716,31.211,155.927
C02519=1048.828,-117.748,431.932,169.713,31.210,155.927
C02520=1048.822,-117.998,431.942,169.711,31.210,155.927
C02521=1048.815,-118.248,431.951,169.709,31.210,155.927
C02522=1048.809,-118.498,431.961,169.706,31.209,155.927
C02523=1048.803,-118.748,431.970,169.704,31.209,155.927
C02524=1048.798,-118.997,431.980,169.702,31.209,155.927
C02525=1048.791,-119.246,431.989,169.700,31.208,155.927
C02526=1048.785,-119.497,431.997,169.698,31.208,155.927
C02527=1048.779,-119.746,432.007,169.696,31.208,155.927
C02528=1048.772,-119.996,432.017,169.694,31.208,155.927
C02529=1048.766,-120.246,432.026,169.692,31.208,155.928
C02530=1048.761,-120.495,432.035,169.689,31.207,155.928
C02531=1048.755,-120.745,432.045,169.687,31.207,155.928
C02532=1048.749,-120.995,432.054,169.685,31.207,155.928
C02533=1048.742,-121.245,432.063,169.682,31.206,155.928
C02534=1048.736,-121.495,432.072,169.680,31.206,155.928
C02535=1048.729,-121.744,432.082,169.678,31.206,155.928
C02536=1048.724,-121.993,432.091,169.676,31.206,155.928
C02537=1048.718,-122.244,432.100,169.673,31.206,155.928
C02538=1048.712,-122.494,432.109,169.671,31.205,155.928
C02539=1048.706,-122.743,432.119,169.669,31.205,155.928
C02540=1048.699,-122.993,432.128,169.666,31.205,155.929
C02541=1048.693,-123.243,432.136,169.664,31.205,155.929
C02542=1048.687,-123.492,432.146,169.662,31.205,155.929
C02543=1048.681,-123.742,432.156,169.660,31.204,155.929
C02544=1048.675,-123.993,432.164,169.658,31.204,155.929
C02545=1048.669,-124.241,432.173,169.656,31.204,155.929
C02546=1048.663,-124.491,432.183,169.654,31.204,155.929
C02547=1048.657,-124.741,432.192,169.652,31.204,155.929
C02548=1048.651,-124.991,432.201,169.649,31.203,155.929
C02549=1048.644,-125.240,432.210,169.647,31.204,155.929
C02550=1048.638,-125.490,432.219,169.645,31.203,155.929
C02551=1048.632,-125.740,432.228,169.642,31.203,155.930
C02552=1048.625,-125.990,432.237,169.640,31.203,155.930
C02553=1048.620,-126.240,432.246,169.638,31.203,155.930
C02554=1048.614,-126.489,432.255,169.635,31.203,155.930
C02555=1048.608,-126.739,432.265,169.633,31.203,155.930
C02556=1048.601,-126.989,432.273,169.631,31.203,155.930
C02557=1048.596,-127.238,432.282,169.629,31.202,155.930
C02558=1048.590,-127.488,432.292,169.626,31.203,155.930
C02559=1048.583,-127.738,432.300,169.624,31.202,155.930
C02560=1048.577,-127.987,432.309,169.622,31.202,155.930
C02561=1048.573,-128.237,432.320,169.620,31.201,155.930
C02562=1048.570,-128.488,432.330,169.618,31.200,155.930
C02563=1048.567,-128.738,432.341,169.617,31.198,155.930
C02564=1048.565,-128.987,432.353,169.615,31.196,155.930
C02565=1048.565,-129.238,432.365,169.613,31.193,155.929
C02566=1048.566,-129.488,432.379,169.612,31.190,155.929
C02567=1048.567,-129.739,432.393,169.610,31.186,155.928
C02568=1048.569,-129.988,432.407,169.610,31.182,155.928
C02569=1048.573,-130.240,432.422,169.608,31.177,155.927
C02570=1048.578,-130.490,432.437,169.607,31.172,155.926
C02571=1048.584,-130.741,432.454,169.606,31.167,155.925
C02572=1048.589,-130.990,432.471,169.606,31.160,155.924
C02573=1048.228,-131.014,432.240,169.560,31.333,155.956
C02574=1048.221,-130.764,432.223,169.561,31.339,155.957
C02575=1048.216,-130.514,432.207,169.561,31.344,155.958
C02576=1048.211,-130.264,432.191,169.562,31.350,155.959
C02577=1048.208,-130.012,432.176,169.563,31.354,155.960
C02578=1048.206,-129.763,432.162,169.565,31.359,155.961
C02579=1048.203,-129.512,432.148,169.566,31.362,155.961
C02580=1048.203,-129.261,432.135,169.567,31.365,155.962
C02581=1048.204,-129.011,432.122,169.569,31.368,155.962
C02582=1048.205,-128.761,432.111,169.570,31.370,155.962
C02583=1048.208,-128.511,432.099,169.572,31.372,155.962
C02584=1048.211,-128.261,432.088,169.574,31.373,155.963
C02585=1048.216,-128.011,432.078,169.577,31.374,155.963
C02586=1048.221,-127.761,432.068,169.579,31.375,155.963
C02587=1048.227,-127.512,432.060,169.581,31.375,155.962
C02588=1048.233,-127.262,432.051,169.583,31.375,155.962
C02589=1048.239,-127.013,432.041,169.586,31.375,155.962
C02590=1048.246,-126.763,432.033,169.587,31.375,155.962
C02591=1048.252,-126.513,432.024,169.589,31.375,155.962
C02592=1048.258,-126.263,432.014,169.592,31.375,155.962
C02593=1048.264,-126.014,432.006,169.594,31.376,155.962
C02594=1048.270,-125.764,431.997,169.596,31.375,155.962
C02595=1048.276,-125.514,431.988,169.598,31.376,155.962
C02596=1048.283,-125.264,431.979,169.601,31.376,155.962
C02597=1048.289,-125.015,431.970,169.603,31.376,155.961
C02598=1048.294,-124.765,431.961,169.605,31.376,155.961
C02599=1048.301,-124.515,431.951,169.608,31.376,155.961
C02600=1048.307,-124.265,431.942,169.610,31.376,155.961
C02601=1048.313,-124.016,431.934,169.612,31.376,155.961
C02602=1048.319,-123.766,431.924,169.615,31.377,155.961
C02603=1048.325,-123.516,431.915,169.617,31.377,155.961
C02604=1048.331,-123.266,431.905,169.619,31.377,155.961
C02605=1048.338,-123.016,431.897,169.621,31.377,155.961
C02606=1048.343,-122.767,431.888,169.624,31.377,155.961
C02607=1048.350,-122.517,431.878,169.626,31.378,155.960
C02608=1048.356,-122.268,431.868,169.628,31.378,155.960
C02609=1048.362,-122.017,431.860,169.631,31.378,155.960
C02610=1048.368,-121.767,431.850,169.632,31.378,155.960
C02611=1048.374,-121.519,431.841,169.634,31.378,155.960
C02612=1048.380,-121.269,431.832,169.636,31.378,155.960
C02613=1048.386,-121.018,431.823,169.639,31.379,155.960
C02614=1048.392,-120.769,431.813,169.641,31.379,155.960
C02615=1048.398,-120.519,431.804,169.643,31.379,155.960
C02616=1048.404,-120.270,431.795,169.646,31.379,155.960
C02617=1048.410,-120.020,431.785,169.648,31.380,155.960
C02618=1048.416,-119.770,431.775,169.650,31.380,155.959
C02619=1048.423,-119.520,431.767,169.652,31.380,155.959
C02620=1048.429,-119.270,431.758,169.655,31.380,155.959
C02621=1048.435,-119.020,431.748,169.657,31.380,155.959
C02622=1048.442,-118.771,431.738,169.659,31.380,155.959
C02623=1048.447,-118.521,431.729,169.662,31.381,155.959
C02624=1048.453,-118.272,431.720,169.664,31.381,155.959
C02625=1048.459,-118.022,431.710,169.666,31.381,155.959
C02626=1048.465,-117.771,431.701,169.668,31.382,155.959
C02627=1048.471,-117.522,431.692,169.671,31.382,155.959
C02628=1048.478,-117.272,431.682,169.672,31.382,155.959
C02629=1048.485,-117.022,431.673,169.674,31.383,155.959
C02630=1048.491,-116.773,431.664,169.677,31.383,155.959
C02631=1048.496,-116.523,431.654,169.679,31.383,155.958
C02632=1048.502,-116.274,431.645,169.681,31.384,155.958
C02633=1048.509,-116.024,431.635,169.683,31.384,155.958
C02634=1048.516,-115.738,431.624,169.686,31.384,155.958
C02635=1048.523,-115.453,431.613,169.689,31.385,155.958
C02636=1048.530,-115.168,431.602,169.691,31.385,155.958
C02637=1048.536,-114.883,431.591,169.694,31.385,155.958
C02638=1048.543,-114.633,431.582,169.696,31.386,155.958
C02639=1048.549,-114.383,431.572,169.698,31.386,155.958
C02640=1048.555,-114.133,431.563,169.701,31.386,155.958
C02641=1048.561,-113.883,431.553,169.703,31.387,155.958
C02642=1048.567,-113.634,431.543,169.705,31.387,155.958
C02643=1048.573,-113.384,431.534,169.707,31.387,155.958
C02644=1048.580,-113.134,431.524,169.710,31.388,155.958
C02645=1048.586,-112.884,431.515,169.711,31.388,155.958
C02646=1048.592,-112.634,431.505,169.713,31.388,155.957
C02647=1048.598,-112.385,431.496,169.715,31.388,155.957
C02648=1048.604,-112.135,431.486,169.718,31.389,155.957
C02649=1048.610,-111.885,431.476,169.720,31.390,155.957
C02650=1048.616,-111.635,431.466,169.722,31.390,155.957
C02651=1048.622,-111.385,431.457,169.724,31.390,155.957
C02652=1048.629,-111.136,431.446,169.727,31.391,155.957
C02653=1048.635,-110.886,431.437,169.729,31.391,155.957
C02654=1048.641,-110.636,431.427,169.731,31.391,155.957
C02655=1048.647,-110.387,431.418,169.734,31.392,155.957
C02656=1048.653,-110.137,431.408,169.736,31.392,155.957
C02657=1048.659,-109.887,431.399,169.738,31.393,155.957
C02658=1048.666,-109.638,431.388,169.740,31.393,155.957
C02659=1048.672,-109.388,431.379,169.743,31.394,155.957
C02660=1048.678,-109.138,431.369,169.745,31.394,155.957
C02661=1048.684,-108.888,431.359,169.747,31.394,155.957
C02662=1048.690,-108.638,431.349,169.748,31.395,155.957
C02663=1048.696,-108.389,431.339,169.751,31.395,155.957
C02664=1048.702,-108.139,431.330,169.753,31.396,155.957
C02665=1048.709,-107.890,431.320,169.755,31.396,155.957
C02666=1048.715,-107.640,431.310,169.757,31.396,155.956
C02667=1048.721,-107.390,431.301,169.760,31.397,155.956
C02668=1048.727,-107.140,431.290,169.762,31.398,155.956
C02669=1048.733,-106.891,431.280,169.764,31.398,155.956
C02670=1048.739,-106.641,431.271,169.766,31.398,155.956
C02671=1048.746,-106.392,431.261,169.769,31.399,155.956
C02672=1048.751,-106.142,431.250,169.771,31.400,155.956
C02673=1048.757,-105.892,431.241,169.773,31.400,155.956
C02674=1048.764,-105.643,431.231,169.775,31.401,155.956
C02675=1048.770,-105.393,431.221,169.778,31.401,155.956
C02676=1048.775,-105.143,431.211,169.780,31.401,155.956
C02677=1048.782,-104.893,431.200,169.781,31.402,155.956
C02678=1048.788,-104.643,431.191,169.783,31.403,155.956
C02679=1048.795,-104.393,431.181,169.786,31.403,155.956
C02680=1048.800,-104.144,431.170,169.788,31.404,155.956
C02681=1048.807,-103.894,431.161,169.790,31.404,155.956
C02682=1048.813,-103.644,431.151,169.792,31.404,155.956
C02683=1048.818,-103.395,431.140,169.795,31.405,155.956
C02684=1048.825,-103.145,431.131,169.797,31.406,155.956
C02685=1048.831,-102.896,431.120,169.799,31.407,155.956
C02686=1048.837,-102.646,431.111,169.801,31.407,155.956
C02687=1048.843,-102.395,431.100,169.804,31.407,155.956
C02688=1048.850,-102.146,431.090,169.806,31.408,155.956
C02689=1048.856,-101.896,431.080,169.808,31.409,155.956
C02690=1048.862,-101.647,431.070,169.810,31.409,155.956
C02691=1048.868,-101.397,431.060,169.813,31.410,155.956
C02692=1048.874,-101.148,431.050,169.814,31.411,155.956
C02693=1048.880,-100.898,431.040,169.816,31.411,155.956
C02694=1048.887,-100.648,431.029,169.818,31.411,155.956
C02695=1048.893,-100.398,431.019,169.820,31.412,155.956
C02696=1048.899,-100.148,431.008,169.823,31.413,155.956
C02697=1048.905,-99.899,430.999,169.825,31.414,155.956
C02698=1048.912,-99.613,430.987,169.827,31.414,155.956
C02699=1048.919,-99.326,430.975,169.830,31.415,155.956
C02700=1048.926,-99.040,430.963,169.833,31.415,155.956
C02701=1048.933,-98.752,430.952,169.835,31.416,155.956
C02702=1048.940,-98.503,430.942,169.837,31.416,155.956
C02703=1048.945,-98.253,430.931,169.840,31.417,155.956
C02704=1048.952,-98.003,430.921,169.842,31.418,155.956
C02705=1048.959,-97.754,430.911,169.844,31.419,155.956
C02706=1048.964,-97.504,430.900,169.845,31.419,155.956
C02707=1048.971,-97.255,430.890,169.848,31.420,155.956
C02708=1048.976,-97.005,430.880,169.850,31.421,155.956
C02709=1048.983,-96.755,430.869,169.852,31.421,155.956
C02710=1048.989,-96.505,430.858,169.854,31.422,155.956
C02711=1048.994,-96.255,430.848,169.856,31.423,155.956
C02712=1049.001,-96.006,430.838,169.859,31.423,155.956
C02713=1049.006,-95.756,430.827,169.861,31.424,155.956
C02714=1049.013,-95.507,430.818,169.863,31.425,155.956
C02715=1049.019,-95.256,430.806,169.865,31.425,155.956
C02716=1049.025,-95.007,430.795,169.867,31.426,155.956
C02717=1049.031,-94.757,430.786,169.870,31.427,155.956
C02718=1049.037,-94.508,430.775,169.872,31.428,155.956
C02719=1049.044,-94.258,430.764,169.873,31.429,155.956
C02720=1049.049,-94.008,430.753,169.875,31.429,155.956
C02721=1049.055,-93.758,430.743,169.877,31.430,155.956
C02722=1049.061,-93.509,430.733,169.880,31.431,155.956
C02723=1049.068,-93.259,430.722,169.882,31.432,155.956
C02724=1049.074,-93.010,430.711,169.884,31.433,155.956
C02725=1049.080,-92.759,430.701,169.886,31.433,155.956
C02726=1049.085,-92.510,430.690,169.888,31.434,155.956
C02727=1049.092,-92.260,430.680,169.891,31.435,155.956
C02728=1049.098,-92.011,430.669,169.893,31.436,155.956
C02729=1049.105,-91.761,430.659,169.895,31.436,155.956
C02730=1049.110,-91.511,430.648,169.897,31.437,155.956
C02731=1049.116,-91.261,430.637,169.899,31.438,155.956
C02732=1049.123,-91.012,430.627,169.901,31.439,155.956
C02733=1049.129,-90.762,430.616,169.903,31.439,155.956
C02734=1049.135,-90.512,430.605,169.905,31.440,155.956
C02735=1049.141,-90.262,430.595,169.907,31.441,155.956
C02736=1049.147,-90.013,430.584,169.909,31.442,155.956
C02737=1049.153,-89.763,430.573,169.912,31.443,155.956
C02738=1049.160,-89.514,430.563,169.914,31.443,155.956
C02739=1049.165,-89.264,430.552,169.916,31.444,155.956
C02740=1049.172,-89.014,430.541,169.918,31.445,155.956
C02741=1049.178,-88.765,430.530,169.920,31.446,155.956
C02742=1049.184,-88.515,430.520,169.923,31.447,155.956
C02743=1049.191,-88.265,430.509,169.925,31.447,155.956
C02744=1049.196,-88.015,430.499,169.927,31.448,155.956
C02745=1049.202,-87.766,430.488,169.929,31.449,155.956
C02746=1049.209,-87.516,430.477,169.930,31.450,155.956
C02747=1049.215,-87.266,430.466,169.933,31.451,155.956
C02748=1049.221,-87.017,430.455,169.935,31.451,155.956
C02749=1049.228,-86.767,430.445,169.937,31.452,155.956
C02750=1049.234,-86.518,430.434,169.939,31.453,155.956
C02751=1049.240,-86.267,430.423,169.941,31.454,155.956
C02752=1049.246,-86.018,430.412,169.944,31.455,155.956
C02753=1049.252,-85.769,430.402,169.946,31.456,155.957
C02754=1049.259,-85.519,430.390,169.948,31.457,155.957
C02755=1049.264,-85.269,430.379,169.950,31.457,155.957
C02756=1049.271,-85.019,430.369,169.952,31.458,155.957
C02757=1049.277,-84.770,430.358,169.955,31.459,155.957
C02758=1049.283,-84.519,430.347,169.957,31.460,155.957
C02759=1049.290,-84.270,430.336,169.958,31.461,155.957
C02760=1049.296,-84.021,430.325,169.960,31.462,155.957
C02761=1049.302,-83.771,430.314,169.962,31.462,155.957
C02762=1049.309,-83.487,430.302,169.965,31.464,155.957
C02763=1049.316,-83.203,430.289,169.967,31.464,155.957
C02764=1049.324,-82.919,430.277,169.970,31.465,155.957
C02765=1049.331,-82.634,430.265,169.972,31.466,155.957
C02766=1049.337,-82.384,430.254,169.974,31.467,155.957
C02767=1049.343,-82.135,430.242,169.977,31.468,155.957
C02768=1049.350,-81.885,430.231,169.979,31.469,155.957
C02769=1049.356,-81.636,430.221,169.981,31.469,155.957
C02770=1049.362,-81.386,430.209,169.983,31.470,155.957
C02771=1049.368,-81.136,430.198,169.984,31.471,155.957
C02772=1049.375,-80.886,430.188,169.986,31.472,155.957
C02773=1049.381,-80.637,430.177,169.989,31.473,155.957
C02774=1049.387,-80.387,430.165,169.991,31.474,155.957
C02775=1049.393,-80.138,430.154,169.993,31.475,155.957
C02776=1049.400,-79.888,430.143,169.995,31.476,155.957
C02777=1049.406,-79.638,430.133,169.997,31.477,155.957
C02778=1049.412,-79.388,430.121,169.999,31.478,155.958
C02779=1049.418,-79.139,430.110,170.002,31.479,155.958
C02780=1049.425,-78.889,430.098,170.004,31.480,155.958
C02781=1049.430,-78.640,430.088,170.006,31.481,155.958
C02782=1049.437,-78.389,430.076,170.008,31.482,155.958
C02783=1049.443,-78.141,430.065,170.009,31.483,155.958
C02784=1049.449,-77.890,430.054,170.011,31.484,155.958
C02785=1049.455,-77.641,430.043,170.014,31.485,155.958
C02786=1049.461,-77.391,430.031,170.016,31.486,155.958
C02787=1049.468,-77.141,430.019,170.018,31.487,155.958
C02788=1049.473,-76.892,430.009,170.020,31.488,155.958
C02789=1049.480,-76.641,429.997,170.022,31.489,155.958
C02790=1049.486,-76.393,429.986,170.024,31.490,155.958
C02791=1049.492,-76.142,429.974,170.026,31.491,155.958
C02792=1049.498,-75.893,429.964,170.029,31.492,155.958
C02793=1049.505,-75.643,429.952,170.031,31.493,155.958
C02794=1049.510,-75.394,429.941,170.033,31.494,155.959
C02795=1049.517,-75.144,429.930,170.034,31.495,155.959
C02796=1049.523,-74.894,429.918,170.036,31.496,155.959
C02797=1049.529,-74.645,429.907,170.038,31.497,155.959
C02798=1049.536,-74.395,429.896,170.040,31.498,155.959
C02799=1049.542,-74.146,429.884,170.043,31.499,155.959
C02800=1049.548,-73.895,429.873,170.045,31.500,155.959
C02801=1049.554,-73.646,429.861,170.047,31.501,155.959
C02802=1049.560,-73.396,429.850,170.049,31.502,155.959
C02803=1049.566,-73.147,429.838,170.051,31.504,155.959
C02804=1049.573,-72.897,429.827,170.053,31.505,155.959
C02805=1049.578,-72.647,429.814,170.055,31.506,155.959
C02806=1049.584,-72.398,429.804,170.057,31.507,155.960
C02807=1049.591,-72.148,429.792,170.059,31.508,155.960
C02808=1049.597,-71.899,429.781,170.061,31.509,155.960
C02809=1049.602,-71.648,429.769,170.063,31.510,155.960
C02810=1049.608,-71.399,429.757,170.065,31.511,155.960
C02811=1049.615,-71.150,429.745,170.067,31.513,155.960
C02812=1049.621,-70.900,429.734,170.069,31.514,155.960
C02813=1049.627,-70.650,429.722,170.071,31.515,155.960
C02814=1049.633,-70.400,429.711,170.073,31.516,155.960
C02815=1049.639,-70.151,429.699,170.075,31.517,155.960
C02816=1049.645,-69.901,429.688,170.078,31.519,155.961
C02817=1049.651,-69.651,429.675,170.080,31.520,155.961
C02818=1049.657,-69.402,429.664,170.082,31.521,155.961
C02819=1049.664,-69.152,429.652,170.083,31.522,155.961
C02820=1049.670,-68.903,429.640,170.085,31.523,155.961
C02821=1049.675,-68.653,429.629,170.087,31.524,155.961
C02822=1049.682,-68.403,429.617,170.089,31.525,155.961
C02823=1049.688,-68.154,429.606,170.091,31.526,155.961
C02824=1049.694,-67.904,429.594,170.093,31.528,155.961
C02825=1049.700,-67.654,429.582,170.096,31.529,155.961
C02826=1049.707,-67.372,429.569,170.098,31.530,155.961
C02827=1049.714,-67.091,429.556,170.100,31.532,155.962
C02828=1049.721,-66.809,429.542,170.103,31.533,155.962
C02829=1049.728,-66.526,429.529,170.105,31.534,155.962
C02830=1049.735,-66.276,429.517,170.106,31.535,155.962
C02831=1049.740,-66.027,429.505,170.108,31.537,155.962
C02832=1049.746,-65.777,429.494,170.110,31.538,155.962
C02833=1049.753,-65.527,429.482,170.112,31.539,155.962
C02834=1049.758,-65.278,429.470,170.115,31.540,155.962
C02835=1049.764,-65.028,429.458,170.117,31.542,155.962
C02836=1049.771,-64.778,429.446,170.119,31.543,155.963
C02837=1049.778,-64.529,429.434,170.121,31.544,155.963
C02838=1049.783,-64.280,429.422,170.123,31.545,155.963
C02839=1049.789,-64.029,429.411,170.125,31.546,155.963
C02840=1049.796,-63.780,429.399,170.127,31.547,155.963
C02841=1049.801,-63.531,429.387,170.128,31.549,155.963
C02842=1049.808,-63.281,429.375,170.130,31.550,155.963
C02843=1049.814,-63.031,429.364,170.132,31.551,155.963
C02844=1049.820,-62.781,429.351,170.135,31.552,155.963
C02845=1049.827,-62.532,429.339,170.137,31.554,155.964
C02846=1049.833,-62.283,429.328,170.139,31.555,155.964
C02847=1049.839,-62.033,429.315,170.141,31.556,155.964
C02848=1049.845,-61.783,429.304,170.143,31.557,155.964
C02849=1049.852,-61.533,429.292,170.145,31.559,155.964
C02850=1049.857,-61.284,429.280,170.147,31.560,155.964
C02851=1049.864,-61.034,429.268,170.149,31.561,155.964
C02852=1049.870,-60.785,429.256,170.150,31.562,155.964
C02853=1049.876,-60.535,429.243,170.152,31.563,155.964
C02854=1049.883,-60.285,429.231,170.154,31.564,155.965
C02855=1049.889,-60.036,429.220,170.156,31.566,155.965
C02856=1049.895,-59.786,429.208,170.159,31.567,155.965
C02857=1049.901,-59.536,429.196,170.161,31.568,155.965
C02858=1049.908,-59.287,429.184,170.163,31.569,155.965
C02859=1049.914,-59.037,429.171,170.165,31.571,155.965
C02860=1049.920,-58.787,429.159,170.167,31.572,155.965
C02861=1049.927,-58.538,429.147,170.169,31.573,155.965
C02862=1049.932,-58.288,429.135,170.171,31.575,155.965
C02863=1049.939,-58.039,429.123,170.173,31.576,155.966
C02864=1049.945,-57.789,429.111,170.174,31.577,155.966
C02865=1049.952,-57.539,429.099,170.176,31.578,155.966
C02866=1049.958,-57.290,429.087,170.178,31.579,155.966
C02867=1049.964,-57.040,429.074,170.180,31.581,155.966
C02868=1049.971,-56.790,429.062,170.183,31.582,155.966
C02869=1049.977,-56.541,429.050,170.185,31.584,155.966
C02870=1049.983,-56.292,429.038,170.187,31.584,155.966
C02871=1049.989,-56.042,429.026,170.189,31.586,155.967
C02872=1049.995,-55.792,429.014,170.191,31.587,155.967
C02873=1050.002,-55.543,429.002,170.193,31.588,155.967
C02874=1050.009,-55.293,428.990,170.195,31.590,155.967
C02875=1050.015,-55.043,428.977,170.196,31.591,155.967
C02876=1050.021,-54.794,428.965,170.198,31.592,155.967
C02877=1050.027,-54.544,428.953,170.200,31.594,155.967
C02878=1050.034,-54.294,428.941,170.202,31.595,155.967
C02879=1050.040,-54.045,428.929,170.204,31.596,155.968
C02880=1050.046,-53.795,428.916,170.206,31.597,155.968
C02881=1050.053,-53.545,428.904,170.208,31.599,155.968
C02882=1050.059,-53.295,428.892,170.210,31.600,155.968
C02883=1050.066,-53.046,428.880,170.213,31.601,155.968
C02884=1050.072,-52.796,428.868,170.215,31.603,155.968
C02885=1050.078,-52.547,428.854,170.217,31.604,155.968
C02886=1050.085,-52.297,428.842,170.219,31.605,155.968
C02887=1050.091,-52.047,428.830,170.220,31.606,155.969
C02888=1050.098,-51.798,428.818,170.222,31.608,155.969
C02889=1050.103,-51.548,428.805,170.224,31.609,155.969
C02890=1050.111,-51.268,428.792,170.226,31.610,155.969
C02891=1050.118,-50.987,428.778,170.229,31.612,155.969
C02892=1050.125,-50.706,428.764,170.231,31.613,155.969
C02893=1050.132,-50.426,428.750,170.233,31.615,155.969
C02894=1050.138,-50.176,428.738,170.235,31.617,155.970
C02895=1050.145,-49.926,428.726,170.237,31.617,155.970
C02896=1050.151,-49.677,428.713,170.239,31.619,155.970
C02897=1050.157,-49.427,428.700,170.240,31.620,155.970
C02898=1050.163,-49.177,428.687,170.242,31.622,155.970
C02899=1050.169,-48.928,428.675,170.244,31.623,155.970
C02900=1050.175,-48.678,428.662,170.246,31.625,155.970
C02901=1050.181,-48.429,428.650,170.248,31.626,155.971
C02902=1050.187,-48.179,428.637,170.250,31.628,155.971
C02903=1050.194,-47.930,428.624,170.252,31.629,155.971
C02904=1050.200,-47.680,428.612,170.254,31.630,155.971
C02905=1050.206,-47.430,428.599,170.256,31.632,155.971
C02906=1050.212,-47.181,428.586,170.258,31.633,155.971
C02907=1050.218,-46.931,428.573,170.260,31.635,155.972
C02908=1050.225,-46.681,428.562,170.261,31.636,155.972
C02909=1050.231,-46.432,428.548,170.263,31.638,155.972
C02910=1050.237,-46.182,428.536,170.265,31.639,155.972
C02911=1050.243,-45.932,428.523,170.268,31.641,155.972
C02912=1050.250,-45.683,428.510,170.270,31.642,155.972
C02913=1050.256,-45.433,428.498,170.272,31.644,155.973
C02914=1050.262,-45.183,428.485,170.274,31.645,155.973
C02915=1050.268,-44.934,428.472,170.276,31.646,155.973
C02916=1050.274,-44.685,428.460,170.278,31.648,155.973
C02917=1050.281,-44.435,428.447,170.280,31.649,155.973
C02918=1050.287,-44.185,428.434,170.282,31.651,155.973
C02919=1050.293,-43.936,428.421,170.283,31.652,155.973
C02920=1050.299,-43.686,428.408,170.285,31.654,155.974
C02921=1050.306,-43.436,428.396,170.287,31.655,155.974
C02922=1050.312,-43.187,428.383,170.289,31.657,155.974
C02923=1050.318,-42.937,428.370,170.291,31.658,155.974
C02924=1050.324,-42.688,428.357,170.293,31.660,155.974
C02925=1050.330,-42.438,428.345,170.295,31.661,155.974
C02926=1050.337,-42.189,428.332,170.297,31.663,155.975
C02927=1050.343,-41.939,428.319,170.299,31.664,155.975
C02928=1050.349,-41.690,428.306,170.301,31.666,155.975
C02929=1050.355,-41.440,428.293,170.303,31.667,155.975
C02930=1050.362,-41.190,428.280,170.304,31.669,155.975
C02931=1050.368,-40.940,428.267,170.306,31.670,155.975
C02932=1050.375,-40.691,428.255,170.308,31.671,155.976
C02933=1050.381,-40.441,428.242,170.310,31.673,155.976
C02934=1050.387,-40.192,428.229,170.312,31.674,155.976
C02935=1050.393,-39.943,428.216,170.314,31.676,155.976
C02936=1050.399,-39.693,428.203,170.316,31.677,155.976
C02937=1050.406,-39.443,428.189,170.318,31.679,155.976
C02938=1050.413,-39.193,428.177,170.320,31.680,155.977
C02939=1050.419,-38.944,428.164,170.322,31.682,155.977
C02940=1050.425,-38.695,428.151,170.324,31.683,155.977
C02941=1050.431,-38.445,428.138,170.325,31.685,155.977
C02942=1050.437,-38.195,428.125,170.326,31.687,155.977
C02943=1050.443,-37.946,428.112,170.328,31.688,155.978
C02944=1050.450,-37.696,428.099,170.330,31.690,155.978
C02945=1050.456,-37.446,428.086,170.332,31.691,155.978
C02946=1050.462,-37.196,428.073,170.334,31.693,155.978
C02947=1050.468,-36.947,428.060,170.336,31.694,155.978
C02948=1050.474,-36.698,428.046,170.338,31.696,155.978
C02949=1050.480,-36.448,428.034,170.340,31.698,155.979
C02950=1050.486,-36.198,428.020,170.342,31.699,155.979
C02951=1050.493,-35.949,428.006,170.344,31.701,155.979
C02952=1050.499,-35.699,427.993,170.345,31.702,155.979
C02953=1050.505,-35.449,427.981,170.347,31.704,155.979
C02954=1050.512,-35.169,427.966,170.349,31.706,155.980
C02955=1050.519,-34.889,427.951,170.352,31.708,155.980
C02956=1050.526,-34.609,427.936,170.354,31.709,155.980
C02957=1050.533,-34.329,427.921,170.356,31.711,155.980
C02958=1050.540,-34.079,427.908,170.358,31.713,155.980
C02959=1050.545,-33.829,427.895,170.360,31.714,155.981
C02960=1050.551,-33.580,427.881,170.362,31.716,155.981
C02961=1050.557,-33.330,427.868,170.364,31.717,155.981
C02962=1050.564,-33.081,427.855,170.365,31.719,155.981
C02963=1050.570,-32.831,427.841,170.367,31.721,155.981
C02964=1050.576,-32.581,427.829,170.369,31.722,155.982
C02965=1050.583,-32.332,427.815,170.371,31.724,155.982
C02966=1050.589,-32.083,427.802,170.372,31.725,155.982
C02967=1050.596,-31.833,427.789,170.374,31.727,155.982
C02968=1050.602,-31.583,427.775,170.376,31.729,155.982
C02969=1050.607,-31.334,427.761,170.378,31.730,155.983
C02970=1050.613,-31.085,427.748,170.380,31.732,155.983
C02971=1050.620,-30.834,427.735,170.382,31.733,155.983
C02972=1050.626,-30.585,427.722,170.384,31.735,155.983
C02973=1050.632,-30.336,427.709,170.386,31.737,155.983
C02974=1050.639,-30.086,427.695,170.387,31.738,155.984
C02975=1050.645,-29.836,427.682,170.389,31.740,155.984
C02976=1050.652,-29.587,427.668,170.391,31.741,155.984
C02977=1050.658,-29.338,427.655,170.393,31.743,155.984
C02978=1050.664,-29.087,427.641,170.395,31.745,155.984
C02979=1050.670,-28.838,427.628,170.397,31.746,155.985
C02980=1050.676,-28.589,427.614,170.399,31.748,155.985
C02981=1050.683,-28.339,427.601,170.401,31.749,155.985
C02982=1050.689,-28.090,427.588,170.403,31.751,155.985
C02983=1050.696,-27.840,427.574,170.405,31.753,155.985
C02984=1050.702,-27.591,427.561,170.406,31.754,155.986
C02985=1050.709,-27.341,427.547,170.407,31.756,155.986
C02986=1050.714,-27.092,427.533,170.409,31.757,155.986
C02987=1050.721,-26.842,427.520,170.411,31.759,155.986
C02988=1050.727,-26.592,427.507,170.413,31.761,155.986
C02989=1050.733,-26.343,427.493,170.415,31.762,155.986
C02990=1050.739,-26.093,427.479,170.417,31.765,155.987
C02991=1050.746,-25.844,427.466,170.419,31.766,155.987
C02992=1050.751,-25.594,427.452,170.421,31.768,155.987
C02993=1050.758,-25.344,427.438,170.423,31.770,155.987
C02994=1050.764,-25.095,427.425,170.425,31.771,155.988
C02995=1050.770,-24.845,427.411,170.427,31.773,155.988
C02996=1050.776,-24.595,427.398,170.427,31.775,155.988
C02997=1050.783,-24.346,427.384,170.429,31.776,155.988
C02998=1050.788,-24.096,427.370,170.431,31.778,155.989
C02999=1050.795,-23.846,427.357,170.433,31.780,155.989
C03000=1050.801,-23.598,427.342,170.435,31.781,155.989
C03001=1050.807,-23.348,427.329,170.437,31.783,155.989
C03002=1050.814,-23.098,427.315,170.439,31.785,155.989
C03003=1050.819,-22.849,427.301,170.441,31.786,155.989
C03004=1050.826,-22.599,427.288,170.443,31.788,155.990
C03005=1050.832,-22.349,427.275,170.445,31.790,155.990
C03006=1050.838,-22.101,427.260,170.446,31.792,155.990
C03007=1050.845,-21.851,427.246,170.447,31.793,155.990
C03008=1050.850,-21.601,427.232,170.449,31.795,155.991
C03009=1050.857,-21.352,427.219,170.451,31.797,155.991
C03010=1050.863,-21.102,427.206,170.453,31.798,155.991
C03011=1050.869,-20.853,427.191,170.455,31.800,155.991
C03012=1050.876,-20.603,427.177,170.457,31.802,155.992
C03013=1050.881,-20.353,427.163,170.459,31.803,155.992
C03014=1050.888,-20.103,427.150,170.461,31.806,155.992
C03015=1050.895,-19.855,427.136,170.463,31.807,155.992
C03016=1050.900,-19.605,427.122,170.464,31.809,155.992
C03017=1050.907,-19.355,427.108,170.466,31.811,155.993
C03018=1050.914,-19.074,427.093,170.467,31.813,155.993
C03019=1050.921,-18.793,427.077,170.470,31.814,155.993
C03020=1050.928,-18.512,427.061,170.472,31.816,155.993
C03021=1050.935,-18.231,427.045,170.474,31.818,155.994
C03022=1050.941,-17.981,427.032,170.476,31.820,155.994
C03023=1050.947,-17.732,427.017,170.478,31.822,155.994
C03024=1050.954,-17.483,427.004,170.480,31.824,155.994
C03025=1050.960,-17.233,426.990,170.481,31.825,155.995
C03026=1050.966,-16.984,426.976,170.483,31.827,155.995
C03027=1050.973,-16.734,426.962,170.485,31.828,155.995
C03028=1050.978,-16.484,426.948,170.487,31.831,155.995
C03029=1050.986,-16.235,426.934,170.488,31.832,155.995
C03030=1050.991,-15.985,426.920,170.490,31.834,155.996
C03031=1050.998,-15.735,426.906,170.492,31.836,155.996
C03032=1051.004,-15.487,426.892,170.494,31.837,155.996
C03033=1051.010,-15.236,426.878,170.495,31.839,155.996
C03034=1051.016,-14.987,426.864,170.497,31.841,155.997
C03035=1051.023,-14.737,426.850,170.499,31.843,155.997
C03036=1051.029,-14.488,426.835,170.501,31.845,155.997
C03037=1051.035,-14.238,426.821,170.503,31.846,155.997
C03038=1051.041,-13.989,426.808,170.505,31.848,155.998
C03039=1051.048,-13.739,426.793,170.507,31.850,155.998
C03040=1051.054,-13.490,426.780,170.507,31.852,155.998
C03041=1051.060,-13.240,426.765,170.509,31.853,155.998
C03042=1051.066,-12.991,426.751,170.511,31.855,155.999
C03043=1051.073,-12.741,426.736,170.513,31.857,155.999
C03044=1051.078,-12.492,426.723,170.515,31.859,155.999
C03045=1051.085,-12.242,426.708,170.517,31.861,155.999
C03046=1051.091,-11.992,426.693,170.519,31.863,155.999
C03047=1051.097,-11.743,426.679,170.520,31.865,156.000
C03048=1051.103,-11.493,426.665,170.522,31.866,156.000
C03049=1051.109,-11.244,426.651,170.524,31.868,156.000
C03050=1051.116,-10.995,426.636,170.526,31.870,156.000
C03051=1051.122,-10.745,426.622,170.527,31.872,156.001
C03052=1051.128,-10.495,426.607,170.529,31.874,156.001
C03053=1051.134,-10.246,426.594,170.530,31.875,156.001
C03054=1051.141,-9.996,426.579,170.532,31.877,156.001
C03055=1051.147,-9.746,426.565,170.534,31.879,156.002
C03056=1051.153,-9.498,426.551,170.536,31.881,156.002
C03057=1051.160,-9.248,426.536,170.538,31.883,156.002
C03058=1051.165,-8.998,426.522,170.540,31.884,156.002
C03059=1051.171,-8.749,426.507,170.542,31.886,156.003
C03060=1051.178,-8.500,426.493,170.543,31.888,156.003
C03061=1051.184,-8.250,426.479,170.545,31.890,156.003
C03062=1051.190,-8.000,426.464,170.547,31.892,156.003
C03063=1051.197,-7.751,426.451,170.548,31.894,156.004
C03064=1051.203,-7.501,426.436,170.550,31.896,156.004
C03065=1051.209,-7.251,426.421,170.552,31.897,156.004
C03066=1051.216,-7.003,426.407,170.553,31.899,156.004
C03067=1051.222,-6.753,426.393,170.555,31.901,156.005
C03068=1051.228,-6.504,426.378,170.557,31.903,156.005
C03069=1051.234,-6.254,426.363,170.559,31.905,156.005
C03070=1051.241,-6.004,426.350,170.561,31.906,156.005
C03071=1051.247,-5.755,426.335,170.563,31.908,156.006
C03072=1051.253,-5.505,426.320,170.564,31.910,156.006
C03073=1051.259,-5.255,426.306,170.566,31.912,156.006
C03074=1051.266,-5.006,426.292,170.568,31.914,156.006
C03075=1051.272,-4.757,426.277,170.569,31.915,156.007
C03076=1051.279,-4.507,426.262,170.571,31.917,156.007
C03077=1051.284,-4.258,426.248,170.573,31.920,156.007
C03078=1051.291,-4.008,426.234,170.574,31.921,156.007
C03079=1051.298,-3.759,426.219,170.576,31.923,156.008
C03080=1051.303,-3.510,426.204,170.578,31.924,156.008
C03081=1051.310,-3.260,426.189,170.580,31.927,156.008
C03082=1051.317,-2.976,426.173,170.582,31.929,156.008
C03083=1051.324,-2.694,426.156,170.584,31.931,156.009
C03084=1051.330,-2.412,426.139,170.586,31.933,156.009
C03085=1051.337,-2.129,426.123,170.588,31.935,156.009
C03086=1051.344,-1.879,426.108,170.589,31.937,156.010
C03087=1051.350,-1.630,426.094,170.591,31.939,156.010
C03088=1051.356,-1.380,426.079,170.592,31.941,156.010
C03089=1051.362,-1.131,426.064,170.594,31.943,156.010
C03090=1051.368,-0.882,426.049,170.596,31.945,156.011
C03091=1051.375,-0.632,426.034,170.598,31.947,156.011
C03092=1051.381,-0.383,426.019,170.600,31.949,156.011
C03093=1051.387,-0.134,426.005,170.601,31.951,156.011
C03094=1051.393,0.116,425.990,170.603,31.953,156.012
C03095=1051.399,0.366,425.975,170.605,31.955,156.012
C03096=1051.405,0.615,425.961,170.607,31.956,156.012
C03097=1051.411,0.865,425.946,170.608,31.958,156.013
C03098=1051.417,1.115,425.930,170.609,31.960,156.013
C03099=1051.423,1.364,425.916,170.611,31.963,156.013
C03100=1051.429,1.614,425.901,170.613,31.965,156.013
C03101=1051.436,1.863,425.886,170.615,31.966,156.014
C03102=1051.442,2.113,425.871,170.616,31.968,156.014
C03103=1051.448,2.362,425.856,170.618,31.970,156.014
C03104=1051.454,2.611,425.841,170.620,31.972,156.014
C03105=1051.460,2.861,425.827,170.622,31.974,156.015
C03106=1051.466,3.110,425.812,170.624,31.976,156.015
C03107=1051.473,3.360,425.797,170.625,31.978,156.015
C03108=1051.479,3.609,425.782,170.627,31.980,156.016
C03109=1051.486,3.858,425.766,170.629,31.982,156.016
C03110=1051.491,4.107,425.752,170.630,31.983,156.016
C03111=1051.498,4.357,425.737,170.631,31.985,156.016
C03112=1051.503,4.607,425.721,170.633,31.987,156.017
C03113=1051.510,4.857,425.706,170.635,31.990,156.017
C03114=1051.516,5.106,425.691,170.637,31.992,156.017
C03115=1051.522,5.355,425.677,170.639,31.993,156.017
C03116=1051.528,5.605,425.662,170.640,31.995,156.018
C03117=1051.535,5.855,425.647,170.642,31.997,156.018
C03118=1051.541,6.104,425.632,170.644,31.999,156.018
C03119=1051.548,6.354,425.617,170.646,32.001,156.019
C03120=1051.554,6.602,425.602,170.647,32.003,156.019
C03121=1051.560,6.852,425.587,170.649,32.005,156.019
C03122=1051.566,7.102,425.572,170.650,32.007,156.019
C03123=1051.572,7.352,425.556,170.652,32.009,156.020
C03124=1051.578,7.601,425.541,170.654,32.011,156.020
C03125=1051.585,7.851,425.526,170.655,32.013,156.020
C03126=1051.591,8.099,425.511,170.657,32.014,156.020
C03127=1051.597,8.349,425.496,170.659,32.016,156.021
C03128=1051.604,8.599,425.481,170.661,32.019,156.021
C03129=1051.610,8.848,425.466,170.662,32.021,156.021
C03130=1051.616,9.098,425.451,170.664,32.023,156.022
C03131=1051.622,9.347,425.435,170.666,32.024,156.022
C03132=1051.629,9.597,425.420,170.668,32.026,156.022
C03133=1051.635,9.846,425.406,170.670,32.028,156.022
C03134=1051.641,10.095,425.391,170.670,32.030,156.023
C03135=1051.648,10.344,425.375,170.672,32.032,156.023
C03136=1051.654,10.594,425.360,170.674,32.034,156.023
C03137=1051.660,10.844,425.345,170.676,32.036,156.023
C03138=1051.666,11.094,425.330,170.677,32.038,156.024
C03139=1051.673,11.343,425.314,170.679,32.040,156.024
C03140=1051.679,11.592,425.299,170.681,32.042,156.024
C03141=1051.686,11.842,425.284,170.683,32.043,156.025
C03142=1051.692,12.090,425.269,170.684,32.045,156.025
C03143=1051.698,12.340,425.254,170.686,32.047,156.025
C03144=1051.704,12.590,425.239,170.688,32.050,156.025
C03145=1051.710,12.839,425.223,170.690,32.052,156.026
C03146=1051.719,13.124,425.205,170.692,32.054,156.026
C03147=1051.726,13.409,425.188,170.693,32.056,156.026
C03148=1051.732,13.693,425.171,170.695,32.058,156.027
C03149=1051.739,13.978,425.154,170.697,32.060,156.027
C03150=1051.746,14.227,425.139,170.698,32.062,156.027
C03151=1051.752,14.477,425.122,170.700,32.064,156.028
C03152=1051.758,14.726,425.107,170.702,32.066,156.028
C03153=1051.765,14.975,425.092,170.704,32.068,156.028
C03154=1051.770,15.225,425.076,170.705,32.070,156.028
C03155=1051.777,15.475,425.061,170.707,32.072,156.029
C03156=1051.783,15.724,425.045,170.709,32.074,156.029
C03157=1051.789,15.974,425.030,170.711,32.076,156.029
C03158=1051.796,16.223,425.014,170.712,32.078,156.030
C03159=1051.801,16.473,424.999,170.713,32.080,156.030
C03160=1051.808,16.722,424.983,170.715,32.082,156.030
C03161=1051.814,16.972,424.968,170.717,32.085,156.030
C03162=1051.821,17.221,424.952,170.718,32.086,156.031
C03163=1051.827,17.471,424.937,170.720,32.088,156.031
C03164=1051.832,17.719,424.921,170.722,32.090,156.031
C03165=1051.839,17.969,424.906,170.724,32.092,156.032
C03166=1051.845,18.218,424.890,170.725,32.094,156.032
C03167=1051.851,18.468,424.875,170.727,32.096,156.032
C03168=1051.858,18.717,424.859,170.729,32.098,156.032
C03169=1051.863,18.967,424.844,170.730,32.100,156.033
C03170=1051.870,19.216,424.828,170.732,32.102,156.033
C03171=1051.876,19.466,424.813,170.734,32.104,156.033
C03172=1051.882,19.715,424.797,170.735,32.106,156.034
C03173=1051.889,19.964,424.781,170.736,32.108,156.034
C03174=1051.895,20.214,424.766,170.738,32.110,156.034
C03175=1051.901,20.463,424.750,170.740,32.112,156.035
C03176=1051.907,20.713,424.734,170.742,32.115,156.035
C03177=1051.913,20.962,424.718,170.743,32.116,156.035
C03178=1051.920,21.211,424.703,170.745,32.119,156.035
C03179=1051.925,21.461,424.687,170.747,32.121,156.036
C03180=1051.932,21.710,424.671,170.748,32.123,156.036
C03181=1051.938,21.960,424.655,170.750,32.125,156.036
C03182=1051.944,22.209,424.640,170.752,32.127,156.037
C03183=1051.950,22.459,424.624,170.754,32.129,156.037
C03184=1051.957,22.708,424.608,170.755,32.131,156.037
C03185=1051.963,22.958,424.593,170.757,32.133,156.038
C03186=1051.969,23.207,424.577,170.758,32.135,156.038
C03187=1051.975,23.456,424.561,170.759,32.137,156.038
C03188=1051.981,23.707,424.545,170.761,32.139,156.038
C03189=1051.988,23.956,424.529,170.763,32.141,156.039
C03190=1051.994,24.205,424.513,170.765,32.143,156.039
C03191=1052.001,24.454,424.497,170.766,32.145,156.039
C03192=1052.006,24.704,424.482,170.768,32.147,156.040
C03193=1052.013,24.953,424.466,170.770,32.149,156.040
C03194=1052.019,25.203,424.450,170.771,32.151,156.040
C03195=1052.025,25.452,424.434,170.773,32.153,156.041
C03196=1052.031,25.702,424.419,170.775,32.155,156.041
C03197=1052.037,25.951,424.402,170.777,32.157,156.041
C03198=1052.044,26.200,424.387,170.778,32.159,156.041
C03199=1052.050,26.449,424.370,170.780,32.161,156.042
C03200=1052.056,26.699,424.356,170.781,32.163,156.042
C03201=1052.063,26.949,424.339,170.782,32.165,156.042
C03202=1052.069,27.198,424.323,170.784,32.167,156.043
C03203=1052.076,27.447,424.307,170.786,32.170,156.043
C03204=1052.082,27.697,424.291,170.787,32.171,156.043
C03205=1052.087,27.946,424.274,170.789,32.174,156.044
C03206=1052.094,28.196,424.260,170.791,32.176,156.044
C03207=1052.100,28.445,424.243,170.793,32.178,156.044
C03208=1052.106,28.694,424.227,170.794,32.180,156.045
C03209=1052.112,28.943,424.211,170.796,32.182,156.045
C03210=1052.120,29.230,424.193,170.798,32.184,156.045
C03211=1052.126,29.516,424.174,170.800,32.186,156.046
C03212=1052.133,29.802,424.155,170.802,32.189,156.046
C03213=1052.140,30.087,424.137,170.803,32.191,156.046
C03214=1052.147,30.336,424.121,170.804,32.193,156.047
C03215=1052.153,30.586,424.105,170.806,32.196,156.047
C03216=1052.159,30.836,424.088,170.808,32.198,156.047
C03217=1052.165,31.085,424.072,170.810,32.200,156.048
C03218=1052.171,31.334,424.056,170.811,32.202,156.048
C03219=1052.178,31.583,424.040,170.813,32.204,156.048
C03220=1052.184,31.833,424.024,170.815,32.206,156.048
C03221=1052.190,32.082,424.008,170.816,32.208,156.049
C03222=1052.196,32.332,423.991,170.818,32.210,156.049
C03223=1052.202,32.582,423.975,170.820,32.212,156.049
C03224=1052.209,32.831,423.959,170.821,32.214,156.050
C03225=1052.215,33.080,423.943,170.823,32.217,156.050
C03226=1052.221,33.329,423.927,170.825,32.219,156.050
C03227=1052.227,33.579,423.910,170.826,32.221,156.051
C03228=1052.233,33.828,423.894,170.827,32.223,156.051
C03229=1052.240,34.078,423.878,170.829,32.225,156.051
C03230=1052.246,34.327,423.862,170.830,32.227,156.052
C03231=1052.252,34.576,423.846,170.832,32.229,156.052
C03232=1052.258,34.826,423.829,170.834,32.231,156.052
C03233=1052.264,35.075,423.813,170.836,32.233,156.052
C03234=1052.270,35.325,423.796,170.837,32.235,156.053
C03235=1052.277,35.574,423.781,170.839,32.237,156.053
C03236=1052.283,35.824,423.765,170.841,32.239,156.053
C03237=1052.289,36.073,423.748,170.842,32.242,156.054
C03238=1052.295,36.322,423.731,170.844,32.244,156.054
C03239=1052.302,36.572,423.715,170.846,32.246,156.054
C03240=1052.308,36.821,423.698,170.847,32.248,156.055
C03241=1052.314,37.070,423.683,170.849,32.250,156.055
C03242=1052.320,37.319,423.666,170.851,32.252,156.055
C03243=1052.327,37.569,423.650,170.851,32.254,156.056
C03244=1052.333,37.819,423.634,170.853,32.256,156.056
C03245=1052.339,38.068,423.617,170.855,32.258,156.056
C03246=1052.345,38.317,423.600,170.856,32.260,156.057
C03247=1052.352,38.567,423.584,170.858,32.262,156.057
C03248=1052.358,38.816,423.568,170.860,32.265,156.057
C03249=1052.364,39.065,423.551,170.861,32.266,156.058
C03250=1052.370,39.314,423.534,170.863,32.269,156.058
C03251=1052.376,39.564,423.518,170.865,32.271,156.058
C03252=1052.382,39.814,423.501,170.866,32.273,156.059
C03253=1052.388,40.063,423.485,170.868,32.275,156.059
C03254=1052.394,40.312,423.468,170.870,32.277,156.059
C03255=1052.400,40.562,423.451,170.871,32.279,156.060
C03256=1052.406,40.812,423.435,170.873,32.281,156.060
C03257=1052.413,41.060,423.418,170.875,32.283,156.060
C03258=1052.419,41.310,423.401,170.876,32.286,156.061
C03259=1052.425,41.560,423.385,170.877,32.288,156.061
C03260=1052.431,41.809,423.369,170.879,32.290,156.061
C03261=1052.437,42.058,423.352,170.881,32.292,156.061
C03262=1052.443,42.307,423.335,170.882,32.294,156.062
C03263=1052.450,42.557,423.319,170.884,32.296,156.062
C03264=1052.456,42.806,423.302,170.886,32.299,156.062
C03265=1052.462,43.055,423.286,170.887,32.301,156.063
C03266=1052.469,43.305,423.269,170.889,32.303,156.063
C03267=1052.475,43.554,423.252,170.891,32.305,156.063
C03268=1052.480,43.804,423.235,170.892,32.307,156.064
C03269=1052.486,44.052,423.218,170.894,32.309,156.064
C03270=1052.493,44.302,423.201,170.895,32.311,156.064
C03271=1052.499,44.552,423.185,170.897,32.313,156.065
C03272=1052.504,44.801,423.168,170.899,32.316,156.065
C03273=1052.510,45.050,423.151,170.900,32.318,156.065
C03274=1052.517,45.336,423.131,170.901,32.321,156.066
C03275=1052.525,45.622,423.113,170.903,32.323,156.066
C03276=1052.532,45.908,423.093,170.905,32.325,156.067
C03277=1052.538,46.194,423.073,170.907,32.328,156.067
C03278=1052.545,46.444,423.057,170.909,32.330,156.067
C03279=1052.551,46.692,423.040,170.910,32.333,156.068
C03280=1052.556,46.942,423.023,170.912,32.335,156.068
C03281=1052.562,47.191,423.006,170.914,32.337,156.068
C03282=1052.569,47.441,422.989,170.915,32.339,156.069
C03283=1052.574,47.690,422.972,170.917,32.341,156.069
C03284=1052.580,47.939,422.955,170.919,32.343,156.069
C03285=1052.587,48.189,422.938,170.920,32.345,156.070
C03286=1052.593,48.438,422.922,170.922,32.347,156.070
C03287=1052.599,48.687,422.904,170.924,32.350,156.070
C03288=1052.605,48.937,422.888,170.925,32.352,156.071
C03289=1052.611,49.186,422.871,170.927,32.354,156.071
C03290=1052.617,49.435,422.853,170.927,32.357,156.071
C03291=1052.623,49.685,422.836,170.929,32.359,156.072
C03292=1052.630,49.934,422.819,170.931,32.361,156.072
C03293=1052.636,50.184,422.802,170.932,32.363,156.072
C03294=1052.642,50.433,422.785,170.934,32.365,156.073
C03295=1052.648,50.682,422.769,170.936,32.367,156.073
C03296=1052.654,50.932,422.751,170.937,32.369,156.073
C03297=1052.660,51.180,422.734,170.939,32.371,156.074
C03298=1052.665,51.430,422.717,170.941,32.374,156.074
C03299=1052.672,51.680,422.700,170.942,32.376,156.074
C03300=1052.678,51.928,422.683,170.944,32.378,156.075
C03301=1052.684,52.179,422.666,170.946,32.380,156.075
C03302=1052.691,52.427,422.649,170.947,32.383,156.075
C03303=1052.697,52.676,422.632,170.949,32.385,156.076
C03304=1052.703,52.926,422.615,170.951,32.387,156.076
C03305=1052.709,53.175,422.598,170.952,32.389,156.076
C03306=1052.716,53.425,422.580,170.954,32.391,156.077
C03307=1052.721,53.674,422.563,170.955,32.393,156.077
C03308=1052.728,53.924,422.546,170.956,32.395,156.077
C03309=1052.734,54.172,422.529,170.958,32.397,156.078
C03310=1052.740,54.422,422.511,170.960,32.400,156.078
C03311=1052.746,54.672,422.495,170.961,32.402,156.078
C03312=1052.752,54.921,422.477,170.963,32.404,156.079
C03313=1052.758,55.170,422.460,170.965,32.406,156.079
C03314=1052.764,55.419,422.444,170.966,32.409,156.080
C03315=1052.771,55.669,422.426,170.968,32.411,156.080
C03316=1052.777,55.918,422.409,170.969,32.412,156.080
C03317=1052.783,56.168,422.391,170.971,32.415,156.080
C03318=1052.789,56.416,422.374,170.973,32.417,156.081
C03319=1052.796,56.666,422.357,170.974,32.419,156.081
C03320=1052.801,56.915,422.340,170.976,32.421,156.081
C03321=1052.808,57.165,422.322,170.978,32.423,156.082
C03322=1052.814,57.414,422.305,170.979,32.425,156.082
C03323=1052.820,57.663,422.288,170.981,32.428,156.082
C03324=1052.826,57.913,422.271,170.983,32.430,156.083
C03325=1052.833,58.162,422.253,170.983,32.432,156.083
C03326=1052.839,58.411,422.236,170.985,32.434,156.083
C03327=1052.845,58.661,422.218,170.987,32.436,156.084
C03328=1052.851,58.910,422.201,170.988,32.438,156.084
C03329=1052.858,59.159,422.184,170.990,32.440,156.084
C03330=1052.864,59.409,422.166,170.992,32.443,156.085
C03331=1052.870,59.658,422.150,170.993,32.444,156.085
C03332=1052.876,59.908,422.132,170.995,32.447,156.085
C03333=1052.883,60.157,422.115,170.997,32.449,156.086
C03334=1052.889,60.406,422.098,170.998,32.451,156.086
C03335=1052.895,60.655,422.080,171.000,32.453,156.086
C03336=1052.902,60.904,422.063,171.002,32.455,156.087
C03337=1052.908,61.154,422.045,171.003,32.458,156.087
C03338=1052.915,61.439,422.026,171.005,32.460,156.087
C03339=1052.922,61.725,422.006,171.007,32.462,156.088
C03340=1052.929,62.010,421.985,171.009,32.465,156.088
C03341=1052.936,62.296,421.965,171.011,32.467,156.089
C03342=1052.943,62.546,421.948,171.013,32.469,156.089
C03343=1052.949,62.794,421.931,171.014,32.472,156.089
C03344=1052.955,63.044,421.913,171.015,32.474,156.090
C03345=1052.962,63.293,421.896,171.017,32.476,156.090
C03346=1052.968,63.543,421.878,171.018,32.478,156.090
C03347=1052.975,63.792,421.861,171.020,32.480,156.091
C03348=1052.980,64.041,421.843,171.022,32.482,156.091
C03349=1052.987,64.291,421.826,171.023,32.484,156.091
C03350=1052.993,64.540,421.808,171.025,32.486,156.092
C03351=1052.999,64.789,421.790,171.026,32.488,156.092
C03352=1053.006,65.039,421.773,171.028,32.491,156.092
C03353=1053.011,65.288,421.755,171.030,32.493,156.093
C03354=1053.017,65.538,421.738,171.031,32.495,156.093
C03355=1053.023,65.786,421.721,171.033,32.498,156.093
C03356=1053.030,66.035,421.702,171.035,32.500,156.094
C03357=1053.036,66.285,421.684,171.036,32.502,156.094
C03358=1053.042,66.534,421.667,171.038,32.504,156.094
C03359=1053.048,66.784,421.649,171.040,32.506,156.095
C03360=1053.054,67.033,421.632,171.041,32.508,156.095
C03361=1053.060,67.282,421.614,171.043,32.510,156.095
C03362=1053.067,67.532,421.596,171.045,32.513,156.096
C03363=1053.073,67.780,421.578,171.046,32.515,156.096
C03364=1053.079,68.030,421.560,171.048,32.517,156.096
C03365=1053.085,68.280,421.542,171.049,32.519,156.097
C03366=1053.091,68.528,421.525,171.050,32.521,156.097
C03367=1053.097,68.778,421.507,171.052,32.523,156.097
C03368=1053.103,69.028,421.489,171.053,32.526,156.098
C03369=1053.109,69.276,421.471,171.055,32.528,156.098
C03370=1053.116,69.526,421.454,171.057,32.530,156.098
C03371=1053.122,69.775,421.436,171.058,32.533,156.099
C03372=1053.128,70.025,421.418,171.060,32.535,156.099
C03373=1053.134,70.274,421.400,171.062,32.537,156.100
C03374=1053.140,70.523,421.382,171.063,32.539,156.100
C03375=1053.146,70.772,421.364,171.065,32.541,156.100
C03376=1053.153,71.022,421.347,171.067,32.544,156.101
C03377=1053.158,71.270,421.328,171.068,32.546,156.101
C03378=1053.165,71.520,421.310,171.070,32.548,156.101
C03379=1053.171,71.770,421.293,171.072,32.550,156.102
C03380=1053.177,72.018,421.274,171.073,32.552,156.102
C03381=1053.183,72.268,421.256,171.075,32.554,156.102
C03382=1053.189,72.518,421.238,171.076,32.557,156.103
C03383=1053.195,72.766,421.220,171.078,32.559,156.103
C03384=1053.201,73.016,421.202,171.080,32.561,156.103
C03385=1053.208,73.265,421.185,171.081,32.564,156.104
C03386=1053.213,73.514,421.167,171.083,32.566,156.104
C03387=1053.220,73.763,421.149,171.084,32.568,156.105
C03388=1053.226,74.013,421.131,171.085,32.570,156.105
C03389=1053.232,74.262,421.112,171.087,32.572,156.105
C03390=1053.238,74.511,421.094,171.089,32.575,156.106
C03391=1053.244,74.760,421.076,171.090,32.577,156.106
C03392=1053.250,75.010,421.058,171.092,32.579,156.106
C03393=1053.256,75.259,421.040,171.094,32.581,156.107
C03394=1053.262,75.508,421.022,171.095,32.583,156.107
C03395=1053.268,75.758,421.004,171.097,32.585,156.107
C03396=1053.275,76.007,420.985,171.098,32.588,156.108
C03397=1053.280,76.256,420.968,171.100,32.590,156.108
C03398=1053.287,76.505,420.949,171.102,32.592,156.108
C03399=1053.293,76.755,420.932,171.103,32.594,156.109
C03400=1053.300,77.004,420.913,171.105,32.596,156.109
C03401=1053.305,77.253,420.895,171.107,32.599,156.109
C03402=1053.312,77.539,420.874,171.109,32.601,156.110
C03403=1053.319,77.824,420.853,171.111,32.604,156.110
C03404=1053.326,78.109,420.833,171.112,32.606,156.111
C03405=1053.333,78.395,420.811,171.114,32.609,156.111
C03406=1053.339,78.645,420.794,171.116,32.611,156.111
C03407=1053.346,78.894,420.775,171.118,32.614,156.112
C03408=1053.352,79.143,420.756,171.119,32.616,156.112
C03409=1053.357,79.392,420.739,171.121,32.618,156.113
C03410=1053.364,79.641,420.720,171.121,32.620,156.113
C03411=1053.369,79.891,420.701,171.123,32.622,156.113
C03412=1053.375,80.139,420.683,171.125,32.625,156.114
C03413=1053.382,80.389,420.665,171.126,32.627,156.114
C03414=1053.388,80.638,420.647,171.128,32.629,156.114
C03415=1053.394,80.887,420.628,171.130,32.631,156.115
C03416=1053.399,81.137,420.609,171.131,32.634,156.115
C03417=1053.405,81.386,420.591,171.133,32.636,156.115
C03418=1053.412,81.635,420.573,171.135,32.639,156.116
C03419=1053.418,81.885,420.555,171.136,32.640,156.116
C03420=1053.424,82.134,420.536,171.138,32.642,156.116
C03421=1053.430,82.382,420.518,171.140,32.645,156.117
C03422=1053.435,82.632,420.499,171.141,32.647,156.117
C03423=1053.442,82.881,420.480,171.143,32.650,156.118
C03424=1053.448,83.131,420.462,171.144,32.652,156.118
C03425=1053.454,83.380,420.444,171.146,32.654,156.118
C03426=1053.461,83.629,420.425,171.148,32.656,156.119
C03427=1053.466,83.878,420.406,171.149,32.658,156.119
C03428=1053.472,84.127,420.388,171.151,32.661,156.119
C03429=1053.478,84.377,420.370,171.153,32.663,156.120
C03430=1053.485,84.626,420.351,171.154,32.665,156.120
C03431=1053.491,84.876,420.332,171.156,32.667,156.120
C03432=1053.497,85.125,420.314,171.158,32.669,156.121
C03433=1053.503,85.374,420.296,171.159,32.672,156.121
C03434=1053.509,85.623,420.277,171.161,32.674,156.121
C03435=1053.515,85.872,420.258,171.163,32.677,156.122
C03436=1053.521,86.121,420.239,171.164,32.678,156.122
C03437=1053.527,86.371,420.221,171.165,32.681,156.123
C03438=1053.534,86.620,420.203,171.167,32.683,156.123
C03439=1053.540,86.869,420.184,171.168,32.685,156.123
C03440=1053.545,87.118,420.165,171.170,32.688,156.124
C03441=1053.552,87.367,420.146,171.172,32.690,156.124
C03442=1053.558,87.617,420.128,171.173,32.692,156.124
C03443=1053.564,87.866,420.110,171.175,32.694,156.125
C03444=1053.571,88.115,420.091,171.177,32.696,156.125
C03445=1053.576,88.365,420.072,171.178,32.699,156.126
C03446=1053.583,88.614,420.053,171.180,32.701,156.126
C03447=1053.589,88.863,420.035,171.182,32.703,156.126
C03448=1053.596,89.112,420.016,171.183,32.705,156.127
C03449=1053.601,89.362,419.997,171.185,32.707,156.127
C03450=1053.607,89.611,419.979,171.187,32.709,156.127
C03451=1053.614,89.860,419.960,171.188,32.712,156.128
C03452=1053.620,90.109,419.942,171.190,32.714,156.128
C03453=1053.625,90.358,419.923,171.192,32.717,156.128
C03454=1053.632,90.607,419.904,171.193,32.719,156.129
C03455=1053.637,90.857,419.885,171.195,32.721,156.129
C03456=1053.644,91.106,419.866,171.197,32.723,156.129
C03457=1053.649,91.355,419.847,171.198,32.725,156.130
C03458=1053.656,91.604,419.828,171.200,32.728,156.130
C03459=1053.662,91.854,419.809,171.202,32.730,156.130
C03460=1053.668,92.103,419.790,171.203,32.732,156.131
C03461=1053.674,92.352,419.771,171.205,32.734,156.131
C03462=1053.680,92.602,419.752,171.206,32.737,156.132
C03463=1053.686,92.851,419.733,171.208,32.739,156.132
C03464=1053.692,93.099,419.715,171.210,32.741,156.132
C03465=1053.697,93.349,419.696,171.211,32.743,156.133
C03466=1053.705,93.635,419.675,171.213,32.746,156.133
C03467=1053.712,93.920,419.653,171.214,32.749,156.134
C03468=1053.719,94.205,419.631,171.216,32.751,156.134
C03469=1053.725,94.490,419.609,171.218,32.754,156.134
C03470=1053.731,94.740,419.590,171.220,32.756,156.135
C03471=1053.738,94.988,419.571,171.221,32.758,156.135
C03472=1053.744,95.238,419.552,171.223,32.761,156.136
C03473=1053.750,95.487,419.533,171.225,32.763,156.136
C03474=1053.756,95.736,419.514,171.226,32.766,156.136
C03475=1053.762,95.985,419.495,171.228,32.768,156.137
C03476=1053.768,96.235,419.476,171.230,32.770,156.137
C03477=1053.774,96.484,419.457,171.231,32.772,156.137
C03478=1053.780,96.733,419.438,171.233,32.775,156.138
C03479=1053.787,96.982,419.418,171.235,32.777,156.138
C03480=1053.792,97.231,419.399,171.236,32.779,156.138
C03481=1053.798,97.481,419.380,171.238,32.781,156.139
C03482=1053.804,97.730,419.361,171.240,32.783,156.139
C03483=1053.810,97.979,419.342,171.241,32.786,156.140
C03484=1053.817,98.229,419.323,171.243,32.788,156.140
C03485=1053.823,98.477,419.303,171.245,32.790,156.140
C03486=1053.829,98.726,419.285,171.246,32.792,156.141
C03487=1053.835,98.976,419.266,171.248,32.795,156.141
C03488=1053.841,99.225,419.247,171.250,32.797,156.141
C03489=1053.847,99.474,419.227,171.252,32.799,156.142
C03490=1053.853,99.723,419.208,171.253,32.801,156.142
C03491=1053.859,99.972,419.189,171.255,32.803,156.142
C03492=1053.865,100.223,419.169,171.257,32.806,156.143
C03493=1053.872,100.471,419.150,171.258,32.808,156.143
C03494=1053.878,100.720,419.131,171.260,32.811,156.144
C03495=1053.884,100.970,419.112,171.262,32.813,156.144
C03496=1053.890,101.219,419.093,171.263,32.815,156.144
C03497=1053.896,101.468,419.073,171.265,32.817,156.145
C03498=1053.902,101.717,419.054,171.267,32.820,156.145
C03499=1053.907,101.967,419.035,171.268,32.822,156.145
C03500=1053.914,102.215,419.015,171.270,32.824,156.146
C03501=1053.920,102.465,418.996,171.272,32.826,156.146
C03502=1053.925,102.714,418.977,171.273,32.829,156.147
C03503=1053.931,102.963,418.957,171.275,32.831,156.147
C03504=1053.937,103.212,418.937,171.276,32.833,156.147
C03505=1053.944,103.461,418.918,171.277,32.836,156.148
C03506=1053.950,103.710,418.899,171.279,32.838,156.148
C03507=1053.955,103.960,418.880,171.281,32.841,156.149
C03508=1053.961,104.208,418.860,171.282,32.842,156.149
C03509=1053.968,104.459,418.840,171.284,32.845,156.149
C03510=1053.974,104.707,418.821,171.286,32.847,156.150
C03511=1053.980,104.957,418.801,171.287,32.850,156.150
C03512=1053.986,105.205,418.782,171.289,32.852,156.150
C03513=1053.992,105.455,418.762,171.291,32.854,156.151
C03514=1053.998,105.704,418.742,171.292,32.856,156.151
C03515=1054.003,105.953,418.723,171.294,32.859,156.152
C03516=1054.010,106.202,418.704,171.296,32.861,156.152
C03517=1054.016,106.451,418.684,171.298,32.863,156.152
C03518=1054.021,106.700,418.665,171.299,32.865,156.153
C03519=1054.028,106.950,418.645,171.301,32.868,156.153
C03520=1054.034,107.199,418.626,171.303,32.870,156.153
C03521=1054.040,107.448,418.606,171.304,32.872,156.154
C03522=1054.046,107.697,418.586,171.306,32.874,156.154
C03523=1054.052,107.946,418.567,171.308,32.877,156.155
C03524=1054.058,108.195,418.547,171.309,32.879,156.155
C03525=1054.064,108.445,418.527,171.311,32.882,156.155
C03526=1054.070,108.694,418.508,171.313,32.884,156.156
C03527=1054.076,108.943,418.488,171.315,32.886,156.156
C03528=1054.083,109.192,418.469,171.316,32.888,156.156
C03529=1054.089,109.441,418.450,171.318,32.891,156.157
C03530=1054.096,109.727,418.426,171.320,32.893,156.157
C03531=1054.102,110.012,418.404,171.322,32.896,156.158
C03532=1054.110,110.297,418.382,171.324,32.899,156.158
C03533=1054.116,110.583,418.359,171.326,32.901,156.158
C03534=1054.123,110.832,418.339,171.327,32.903,156.159
C03535=1054.129,111.081,418.320,171.329,32.906,156.159
C03536=1054.135,111.330,418.300,171.331,32.908,156.160
C03537=1054.141,111.579,418.280,171.333,32.910,156.160
C03538=1054.147,111.828,418.261,171.334,32.913,156.160
C03539=1054.153,112.078,418.241,171.336,32.915,156.161
C03540=1054.159,112.327,418.221,171.338,32.917,156.161
C03541=1054.165,112.575,418.201,171.339,32.919,156.161
C03542=1054.171,112.825,418.182,171.341,32.922,156.162
C03543=1054.177,113.074,418.162,171.343,32.924,156.162
C03544=1054.183,113.323,418.141,171.345,32.926,156.163
C03545=1054.189,113.573,418.122,171.346,32.928,156.163
C03546=1054.195,113.821,418.102,171.348,32.931,156.163
C03547=1054.201,114.070,418.082,171.350,32.934,156.164
C03548=1054.206,114.319,418.062,171.351,32.936,156.164
C03549=1054.213,114.569,418.041,171.353,32.938,156.165
C03550=1054.219,114.818,418.022,171.355,32.941,156.165
C03551=1054.225,115.067,418.002,171.357,32.943,156.165
C03552=1054.230,115.316,417.981,171.358,32.945,156.166
C03553=1054.236,115.565,417.961,171.360,32.948,156.166
C03554=1054.243,115.815,417.941,171.362,32.950,156.166
C03555=1054.248,116.063,417.921,171.363,32.952,156.167
C03556=1054.253,116.313,417.901,171.365,32.954,156.167
C03557=1054.259,116.562,417.881,171.366,32.957,156.168
C03558=1054.265,116.811,417.861,171.367,32.959,156.168
C03559=1054.272,117.060,417.841,171.369,32.961,156.168
C03560=1054.277,117.309,417.821,171.371,32.964,156.169
C03561=1054.283,117.558,417.801,171.373,32.967,156.169
C03562=1054.289,117.807,417.781,171.374,32.969,156.170
C03563=1054.296,118.057,417.760,171.376,32.971,156.170
C03564=1054.301,118.306,417.740,171.378,32.974,156.170
C03565=1054.307,118.555,417.720,171.379,32.976,156.171
C03566=1054.313,118.804,417.701,171.381,32.978,156.171
C03567=1054.319,119.053,417.680,171.383,32.981,156.172
C03568=1054.325,119.303,417.660,171.385,32.983,156.172
C03569=1054.331,119.551,417.640,171.386,32.985,156.172
C03570=1054.337,119.800,417.620,171.388,32.987,156.173
C03571=1054.342,120.050,417.599,171.390,32.990,156.173
C03572=1054.348,120.299,417.579,171.392,32.993,156.174
C03573=1054.354,120.548,417.559,171.393,32.994,156.174
C03574=1054.361,120.797,417.539,171.395,32.997,156.174
C03575=1054.366,121.046,417.518,171.397,33.000,156.175
C03576=1054.372,121.295,417.498,171.398,33.002,156.175
C03577=1054.379,121.545,417.478,171.400,33.004,156.176
C03578=1054.384,121.794,417.457,171.402,33.006,156.176
C03579=1054.390,122.043,417.437,171.404,33.009,156.176
C03580=1054.397,122.292,417.417,171.405,33.011,156.177
C03581=1054.402,122.541,417.396,171.407,33.013,156.177
C03582=1054.408,122.789,417.376,171.409,33.016,156.177
C03583=1054.415,123.039,417.355,171.411,33.018,156.178
C03584=1054.421,123.288,417.335,171.412,33.020,156.178
C03585=1054.426,123.537,417.315,171.414,33.023,156.179
C03586=1054.433,123.786,417.295,171.416,33.025,156.179
C03587=1054.439,124.035,417.275,171.418,33.027,156.179
C03588=1054.444,124.284,417.254,171.419,33.030,156.180
C03589=1054.451,124.534,417.234,171.421,33.032,156.180
C03590=1054.457,124.782,417.213,171.423,33.035,156.181
C03591=1054.462,125.031,417.192,171.425,33.037,156.181
C03592=1054.469,125.281,417.172,171.426,33.039,156.181
C03593=1054.475,125.529,417.152,171.428,33.041,156.182
C03594=1054.482,125.815,417.129,171.430,33.044,156.182
C03595=1054.489,126.100,417.105,171.432,33.047,156.183
C03596=1054.496,126.386,417.081,171.434,33.049,156.183
C03597=1054.502,126.670,417.058,171.436,33.052,156.184
C03598=1054.509,126.941,417.036,171.438,33.055,156.184
C03599=1054.515,127.212,417.013,171.440,33.057,156.184
C03600=1054.523,127.483,416.991,171.442,33.060,156.185
C03601=1054.529,127.754,416.969,171.444,33.062,156.185
C03602=1054.534,128.003,416.949,171.446,33.064,156.186
C03603=1054.541,128.252,416.928,171.448,33.067,156.186
C03604=1054.547,128.501,416.908,171.449,33.069,156.186
C03605=1054.553,128.751,416.887,171.451,33.071,156.187
C03606=1054.559,128.999,416.867,171.453,33.073,156.187
C03607=1054.566,129.249,416.846,171.455,33.076,156.187
C03608=1054.571,129.498,416.826,171.456,33.078,156.188
C03609=1054.578,129.747,416.805,171.458,33.081,156.188
C03610=1054.583,129.996,416.784,171.460,33.083,156.189
C03611=1054.590,130.246,416.764,171.462,33.085,156.189
C03612=1054.596,130.494,416.743,171.464,33.088,156.189
C03613=1054.602,130.744,416.722,171.465,33.090,156.190
C03614=1054.608,130.992,416.702,171.467,33.092,156.190
C03615=1054.615,131.241,416.681,171.469,33.094,156.191
C03616=1054.620,131.490,416.661,171.471,33.097,156.191
C03617=1054.627,131.739,416.640,171.473,33.099,156.191
C03618=1054.632,131.988,416.619,171.474,33.101,156.192
C03619=1054.638,132.238,416.598,171.476,33.104,156.192
C03620=1054.644,132.486,416.577,171.478,33.106,156.193
C03621=1054.650,132.736,416.557,171.480,33.108,156.193
C03622=1054.656,132.985,416.535,171.482,33.111,156.193
C03623=1054.662,133.234,416.515,171.483,33.114,156.194
C03624=1054.668,133.483,416.494,171.485,33.116,156.194
C03625=1054.674,133.732,416.474,171.487,33.118,156.195
C03626=1054.680,133.981,416.452,171.489,33.121,156.195
C03627=1054.685,134.230,416.432,171.490,33.123,156.195
C03628=1054.692,134.479,416.411,171.492,33.125,156.196
C03629=1054.698,134.728,416.390,171.494,33.128,156.196
C03630=1054.704,134.977,416.368,171.496,33.130,156.197
C03631=1054.710,135.226,416.348,171.498,33.132,156.197
C03632=1054.716,135.475,416.327,171.499,33.135,156.197
C03633=1054.721,135.724,416.306,171.501,33.137,156.198
C03634=1054.728,135.973,416.285,171.503,33.139,156.198
C03635=1054.733,136.222,416.265,171.505,33.142,156.199
C03636=1054.739,136.471,416.243,171.507,33.145,156.199
C03637=1054.746,136.720,416.222,171.508,33.146,156.199
C03638=1054.752,136.969,416.201,171.510,33.149,156.200
C03639=1054.758,137.219,416.180,171.512,33.152,156.200
C03640=1054.764,137.468,416.160,171.514,33.154,156.201
